// TIA Portal V17 export
// export: Created 2025-07-01T09:58:36.5371957Z, ExportSetting WithDefaults, DisplayName Totally Integrated Automation Portal, DisplayVersion V17 Update 8, DisplayName TIA Portal Openness, DisplayVersion V17 Update 8, DisplayName TIA Portal Version Control Interface, DisplayVersion V17, DisplayName SINAMICS Startdrive Advanced, DisplayVersion V17 SP2, DisplayName SINAMICS Startdrive G110M, G120, G120C, G120D, G120P, G115D, DisplayVersion V17 SP2, DisplayName SINAMICS Startdrive G130, G150, S120, S150, SINAMICS MV, S210, DisplayVersion V17 SP2, DisplayName STEP 7 Professional, DisplayVersion V17 Update 8, DisplayName SINUMERIK ONE STEP 7 Toolbox, DisplayVersion V17 Update 12, DisplayName SINUMERIK ONE PLC Basic Program Plus, DisplayVersion V17 Update 12, DisplayName SINUMERIK 840D sl STEP 7 Toolbox, DisplayVersion V17 Update 12, DisplayName STEP 7 Safety, DisplayVersion V17 Update 6, DisplayName WinCC Advanced, DisplayVersion V17 Update 8
FUNCTION "FC356_NCK_M_CH4_UNIT_2_STA_0" : Void   // FC356, LAD
TITLE = Channel 1 data
{ S7_Optimized_Access := 'FALSE' }
AUTHOR : ETXETAR
VERSION : 1.0
// stored: AutoNumber false, IsIECCheckEnabled false, SetENOAutomatically false, UDAEnableTagReadback false
   VAR_TEMP
      auxm3 : Bool;
      auxm5 : Bool;
   END_VAR
   VAR_TEMP   // added for the SCL form of the ladder/FBD networks
      _w1 : Bool;
      _w2 : Bool;
   END_VAR
BEGIN

REGION Network 1: CALL FB331 M CODE EXTENDED CH1 / M CODE EXTENDED CHANNEL 1
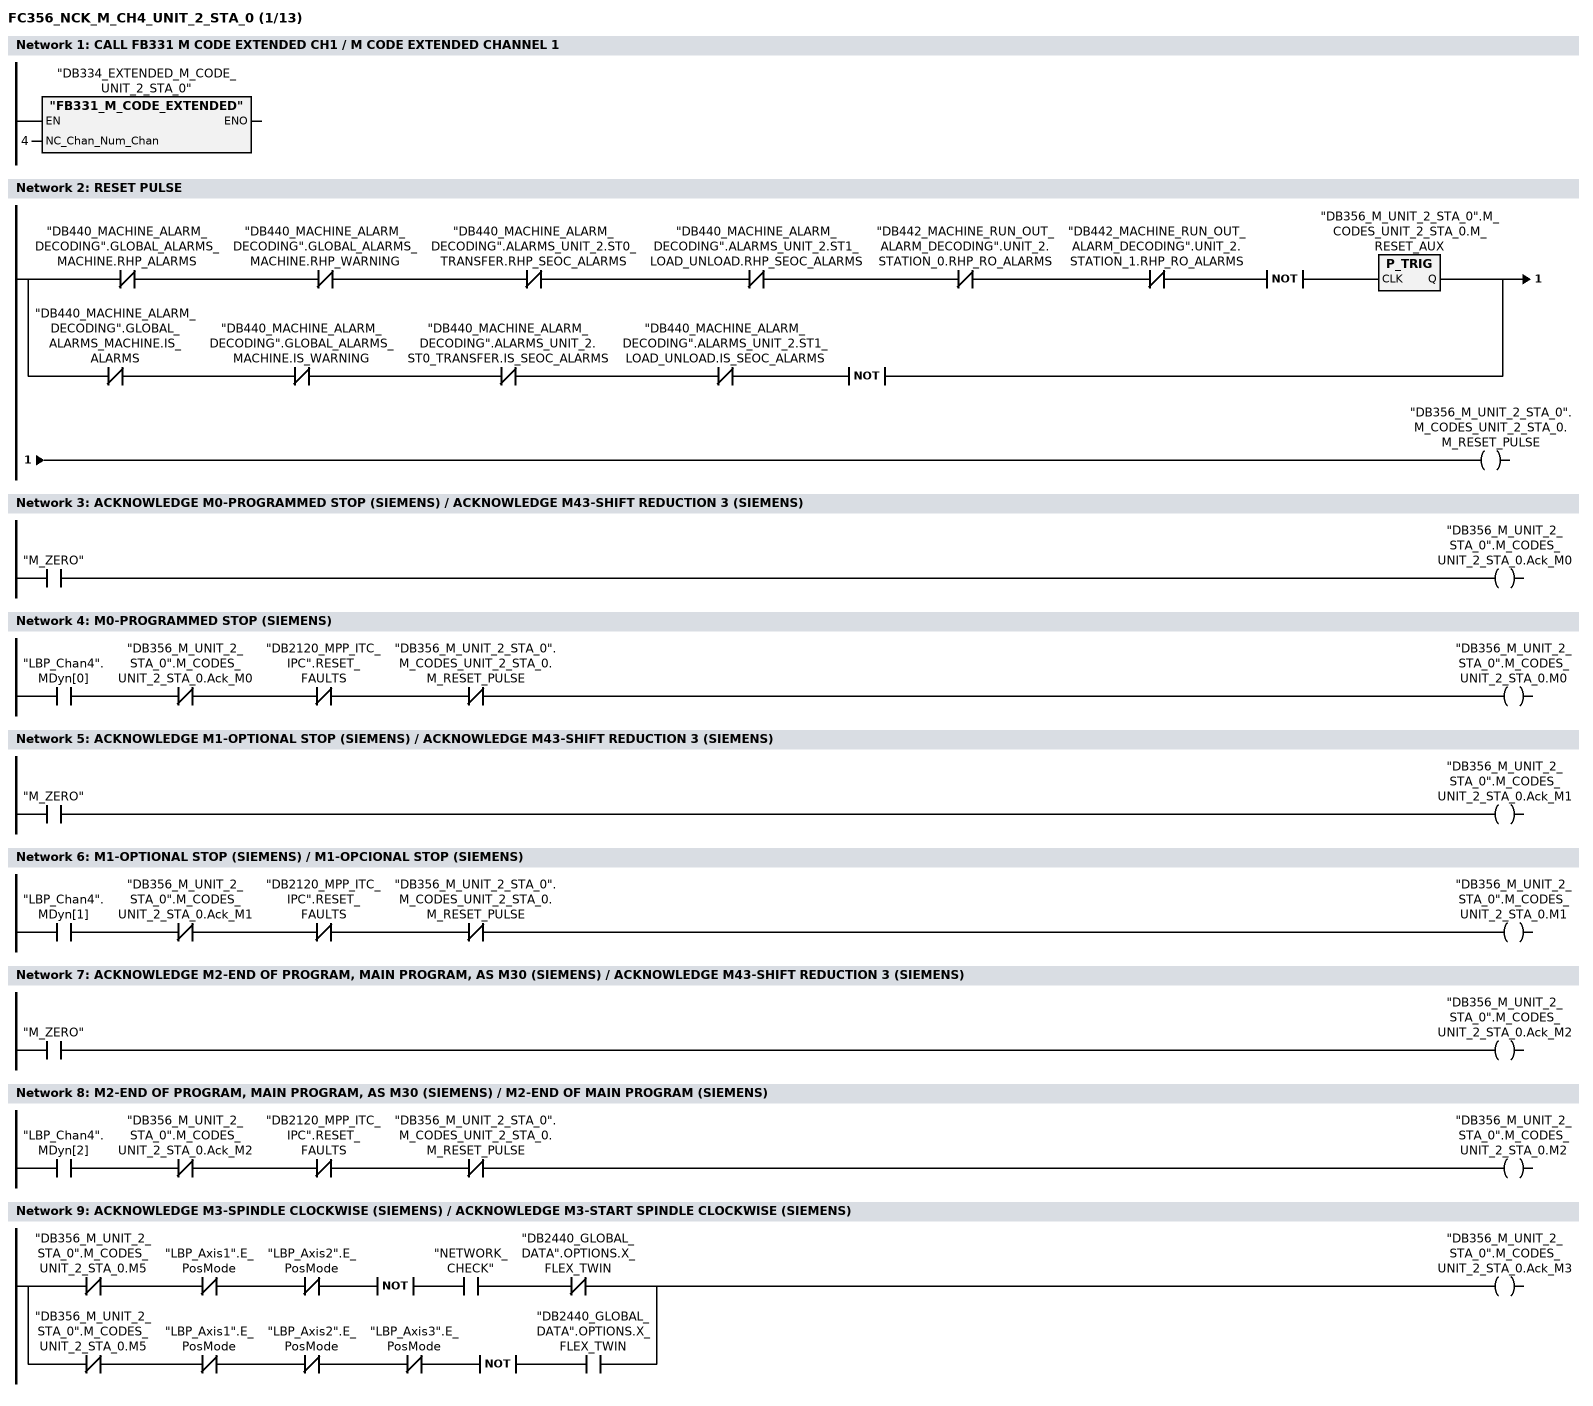
   RUNG wire#powerrail
      "DB334_EXTENDED_M_CODE_UNIT_2_STA_0"(NC_Chan_Num_Chan := 4)
   END_RUNG
   // the same network as SCL:
   "DB334_EXTENDED_M_CODE_UNIT_2_STA_0"(NC_Chan_Num_Chan := 4);   // "FB331_M_CODE_EXTENDED"
END_REGION

REGION Network 2: RESET PULSE
   RUNG wire#powerrail
      I_Contact( "DB440_MACHINE_ALARM_DECODING".GLOBAL_ALARMS_MACHINE.RHP_ALARMS )
      I_Contact( "DB440_MACHINE_ALARM_DECODING".GLOBAL_ALARMS_MACHINE.RHP_WARNING )
      I_Contact( "DB440_MACHINE_ALARM_DECODING".ALARMS_UNIT_2.ST0_TRANSFER.RHP_SEOC_ALARMS )
      I_Contact( "DB440_MACHINE_ALARM_DECODING".ALARMS_UNIT_2.ST1_LOAD_UNLOAD.RHP_SEOC_ALARMS )
      I_Contact( "DB442_MACHINE_RUN_OUT_ALARM_DECODING".UNIT_2.STATION_0.RHP_RO_ALARMS )
      I_Contact( "DB442_MACHINE_RUN_OUT_ALARM_DECODING".UNIT_2.STATION_1.RHP_RO_ALARMS )
      Not()
      P_Trig( "DB356_M_UNIT_2_STA_0".M_CODES_UNIT_2_STA_0.M_RESET_AUX )
      wire#w1
      Coil( "DB356_M_UNIT_2_STA_0".M_CODES_UNIT_2_STA_0.M_RESET_PULSE )
   END_RUNG
   RUNG wire#powerrail
      I_Contact( "DB440_MACHINE_ALARM_DECODING".GLOBAL_ALARMS_MACHINE.IS_ALARMS )
      I_Contact( "DB440_MACHINE_ALARM_DECODING".GLOBAL_ALARMS_MACHINE.IS_WARNING )
      I_Contact( "DB440_MACHINE_ALARM_DECODING".ALARMS_UNIT_2.ST0_TRANSFER.IS_SEOC_ALARMS )
      I_Contact( "DB440_MACHINE_ALARM_DECODING".ALARMS_UNIT_2.ST1_LOAD_UNLOAD.IS_SEOC_ALARMS )
      Not()
   END_RUNG wire#w1
   // the same network as SCL:
   #_w1 := NOT (NOT "DB440_MACHINE_ALARM_DECODING".GLOBAL_ALARMS_MACHINE.RHP_ALARMS AND NOT "DB440_MACHINE_ALARM_DECODING".GLOBAL_ALARMS_MACHINE.RHP_WARNING AND NOT "DB440_MACHINE_ALARM_DECODING".ALARMS_UNIT_2.ST0_TRANSFER.RHP_SEOC_ALARMS AND NOT "DB440_MACHINE_ALARM_DECODING".ALARMS_UNIT_2.ST1_LOAD_UNLOAD.RHP_SEOC_ALARMS AND NOT "DB442_MACHINE_RUN_OUT_ALARM_DECODING".UNIT_2.STATION_0.RHP_RO_ALARMS AND NOT "DB442_MACHINE_RUN_OUT_ALARM_DECODING".UNIT_2.STATION_1.RHP_RO_ALARMS);
   #_w2 := #_w1 AND NOT "DB356_M_UNIT_2_STA_0".M_CODES_UNIT_2_STA_0.M_RESET_AUX;   // rising edge
   "DB356_M_UNIT_2_STA_0".M_CODES_UNIT_2_STA_0.M_RESET_AUX := #_w1;
   "DB356_M_UNIT_2_STA_0".M_CODES_UNIT_2_STA_0.M_RESET_PULSE := #_w2 OR NOT (NOT "DB440_MACHINE_ALARM_DECODING".GLOBAL_ALARMS_MACHINE.IS_ALARMS AND NOT "DB440_MACHINE_ALARM_DECODING".GLOBAL_ALARMS_MACHINE.IS_WARNING AND NOT "DB440_MACHINE_ALARM_DECODING".ALARMS_UNIT_2.ST0_TRANSFER.IS_SEOC_ALARMS AND NOT "DB440_MACHINE_ALARM_DECODING".ALARMS_UNIT_2.ST1_LOAD_UNLOAD.IS_SEOC_ALARMS);
END_REGION

REGION Network 3: ACKNOWLEDGE M0-PROGRAMMED STOP (SIEMENS) / ACKNOWLEDGE M43-SHIFT REDUCTION 3 (SIEMENS)
   RUNG wire#powerrail
      Contact( "M_ZERO" )
      Coil( "DB356_M_UNIT_2_STA_0".M_CODES_UNIT_2_STA_0.Ack_M0 )
   END_RUNG
   // the same network as SCL:
   "DB356_M_UNIT_2_STA_0".M_CODES_UNIT_2_STA_0.Ack_M0 := "M_ZERO";
END_REGION

REGION Network 4: M0-PROGRAMMED STOP (SIEMENS)
   RUNG wire#powerrail
      Contact( "LBP_Chan4".MDyn[0] )
      I_Contact( "DB356_M_UNIT_2_STA_0".M_CODES_UNIT_2_STA_0.Ack_M0 )
      I_Contact( "DB2120_MPP_ITC_IPC".RESET_FAULTS )
      I_Contact( "DB356_M_UNIT_2_STA_0".M_CODES_UNIT_2_STA_0.M_RESET_PULSE )
      Coil( "DB356_M_UNIT_2_STA_0".M_CODES_UNIT_2_STA_0.M0 )
   END_RUNG
   // the same network as SCL:
   "DB356_M_UNIT_2_STA_0".M_CODES_UNIT_2_STA_0.M0 := "LBP_Chan4".MDyn[0] AND NOT "DB356_M_UNIT_2_STA_0".M_CODES_UNIT_2_STA_0.Ack_M0 AND NOT "DB2120_MPP_ITC_IPC".RESET_FAULTS AND NOT "DB356_M_UNIT_2_STA_0".M_CODES_UNIT_2_STA_0.M_RESET_PULSE;
END_REGION

REGION Network 5: ACKNOWLEDGE M1-OPTIONAL STOP (SIEMENS) / ACKNOWLEDGE M43-SHIFT REDUCTION 3 (SIEMENS)
   RUNG wire#powerrail
      Contact( "M_ZERO" )
      Coil( "DB356_M_UNIT_2_STA_0".M_CODES_UNIT_2_STA_0.Ack_M1 )
   END_RUNG
   // the same network as SCL:
   "DB356_M_UNIT_2_STA_0".M_CODES_UNIT_2_STA_0.Ack_M1 := "M_ZERO";
END_REGION

REGION Network 6: M1-OPTIONAL STOP (SIEMENS) / M1-OPCIONAL STOP (SIEMENS)
   RUNG wire#powerrail
      Contact( "LBP_Chan4".MDyn[1] )
      I_Contact( "DB356_M_UNIT_2_STA_0".M_CODES_UNIT_2_STA_0.Ack_M1 )
      I_Contact( "DB2120_MPP_ITC_IPC".RESET_FAULTS )
      I_Contact( "DB356_M_UNIT_2_STA_0".M_CODES_UNIT_2_STA_0.M_RESET_PULSE )
      Coil( "DB356_M_UNIT_2_STA_0".M_CODES_UNIT_2_STA_0.M1 )
   END_RUNG
   // the same network as SCL:
   "DB356_M_UNIT_2_STA_0".M_CODES_UNIT_2_STA_0.M1 := "LBP_Chan4".MDyn[1] AND NOT "DB356_M_UNIT_2_STA_0".M_CODES_UNIT_2_STA_0.Ack_M1 AND NOT "DB2120_MPP_ITC_IPC".RESET_FAULTS AND NOT "DB356_M_UNIT_2_STA_0".M_CODES_UNIT_2_STA_0.M_RESET_PULSE;
END_REGION

REGION Network 7: ACKNOWLEDGE M2-END OF PROGRAM, MAIN PROGRAM, AS M30 (SIEMENS) / ACKNOWLEDGE M43-SHIFT REDUCTION 3 (SIEMENS)
   RUNG wire#powerrail
      Contact( "M_ZERO" )
      Coil( "DB356_M_UNIT_2_STA_0".M_CODES_UNIT_2_STA_0.Ack_M2 )
   END_RUNG
   // the same network as SCL:
   "DB356_M_UNIT_2_STA_0".M_CODES_UNIT_2_STA_0.Ack_M2 := "M_ZERO";
END_REGION

REGION Network 8: M2-END OF PROGRAM, MAIN PROGRAM, AS M30 (SIEMENS) / M2-END OF MAIN PROGRAM (SIEMENS)
   RUNG wire#powerrail
      Contact( "LBP_Chan4".MDyn[2] )
      I_Contact( "DB356_M_UNIT_2_STA_0".M_CODES_UNIT_2_STA_0.Ack_M2 )
      I_Contact( "DB2120_MPP_ITC_IPC".RESET_FAULTS )
      I_Contact( "DB356_M_UNIT_2_STA_0".M_CODES_UNIT_2_STA_0.M_RESET_PULSE )
      Coil( "DB356_M_UNIT_2_STA_0".M_CODES_UNIT_2_STA_0.M2 )
   END_RUNG
   // the same network as SCL:
   "DB356_M_UNIT_2_STA_0".M_CODES_UNIT_2_STA_0.M2 := "LBP_Chan4".MDyn[2] AND NOT "DB356_M_UNIT_2_STA_0".M_CODES_UNIT_2_STA_0.Ack_M2 AND NOT "DB2120_MPP_ITC_IPC".RESET_FAULTS AND NOT "DB356_M_UNIT_2_STA_0".M_CODES_UNIT_2_STA_0.M_RESET_PULSE;
END_REGION

REGION Network 9: ACKNOWLEDGE M3-SPINDLE CLOCKWISE (SIEMENS) / ACKNOWLEDGE M3-START SPINDLE CLOCKWISE (SIEMENS)
   RUNG wire#powerrail
      I_Contact( "DB356_M_UNIT_2_STA_0".M_CODES_UNIT_2_STA_0.M5 )
      I_Contact( "LBP_Axis1".E_PosMode )
      I_Contact( "LBP_Axis2".E_PosMode )
      Not()
      Contact( "NETWORK_CHECK" )
      I_Contact( "DB2440_GLOBAL_DATA".OPTIONS.X_FLEX_TWIN )
      wire#w1
      Coil( "DB356_M_UNIT_2_STA_0".M_CODES_UNIT_2_STA_0.Ack_M3 )
   END_RUNG
   RUNG wire#powerrail
      I_Contact( "DB356_M_UNIT_2_STA_0".M_CODES_UNIT_2_STA_0.M5 )
      I_Contact( "LBP_Axis1".E_PosMode )
      I_Contact( "LBP_Axis2".E_PosMode )
      I_Contact( "LBP_Axis3".E_PosMode )
      Not()
      Contact( "DB2440_GLOBAL_DATA".OPTIONS.X_FLEX_TWIN )
   END_RUNG wire#w1
   // the same network as SCL:
   "DB356_M_UNIT_2_STA_0".M_CODES_UNIT_2_STA_0.Ack_M3 := (NOT (NOT "DB356_M_UNIT_2_STA_0".M_CODES_UNIT_2_STA_0.M5 AND NOT "LBP_Axis1".E_PosMode AND NOT "LBP_Axis2".E_PosMode) AND "NETWORK_CHECK" AND NOT "DB2440_GLOBAL_DATA".OPTIONS.X_FLEX_TWIN) OR (NOT (NOT "DB356_M_UNIT_2_STA_0".M_CODES_UNIT_2_STA_0.M5 AND NOT "LBP_Axis1".E_PosMode AND NOT "LBP_Axis2".E_PosMode AND NOT "LBP_Axis3".E_PosMode) AND "DB2440_GLOBAL_DATA".OPTIONS.X_FLEX_TWIN);
END_REGION

REGION Network 10: M3-SPINDLE CLOCKWISE AUXILIARY (SIEMENS) / Extended address M function 1 (16 bit INT)
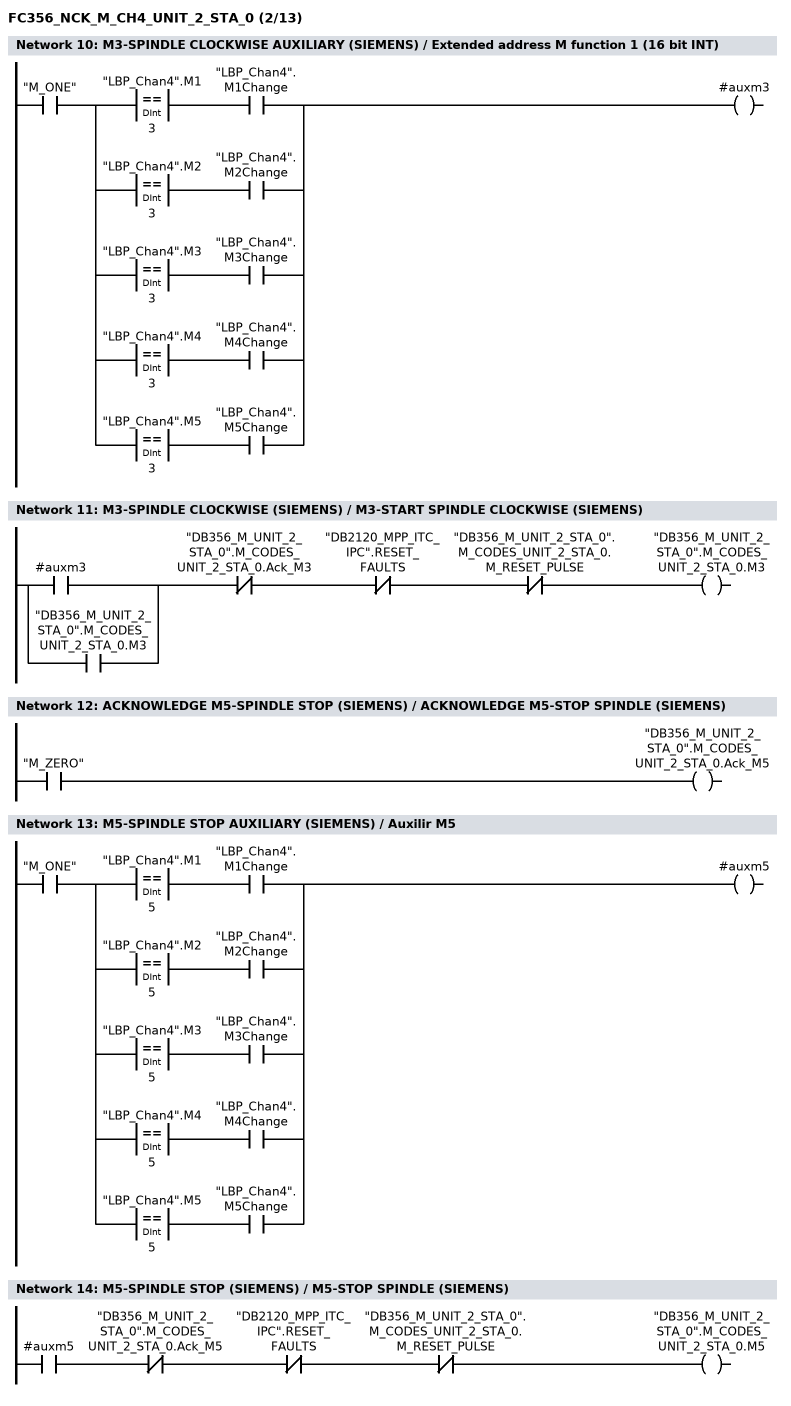
   RUNG wire#powerrail
      Contact( "M_ONE" )
      wire#w1
      { S7_Templates := "SrcType := DInt" } EQ_Contact(in1 := "LBP_Chan4".M1, in2 := 3)
      Contact( "LBP_Chan4".M1Change )
      wire#w2
      Coil( #auxm3 )
   END_RUNG
   RUNG wire#w1
      { S7_Templates := "SrcType := DInt" } EQ_Contact(in1 := "LBP_Chan4".M2, in2 := 3)
      Contact( "LBP_Chan4".M2Change )
   END_RUNG wire#w2
   RUNG wire#w1
      { S7_Templates := "SrcType := DInt" } EQ_Contact(in1 := "LBP_Chan4".M3, in2 := 3)
      Contact( "LBP_Chan4".M3Change )
   END_RUNG wire#w2
   RUNG wire#w1
      { S7_Templates := "SrcType := DInt" } EQ_Contact(in1 := "LBP_Chan4".M4, in2 := 3)
      Contact( "LBP_Chan4".M4Change )
   END_RUNG wire#w2
   RUNG wire#w1
      { S7_Templates := "SrcType := DInt" } EQ_Contact(in1 := "LBP_Chan4".M5, in2 := 3)
      Contact( "LBP_Chan4".M5Change )
   END_RUNG wire#w2
   // the same network as SCL:
   #auxm3 := "M_ONE" AND ((("LBP_Chan4".M1 = 3) AND "LBP_Chan4".M1Change) OR (("LBP_Chan4".M2 = 3) AND "LBP_Chan4".M2Change) OR (("LBP_Chan4".M3 = 3) AND "LBP_Chan4".M3Change) OR (("LBP_Chan4".M4 = 3) AND "LBP_Chan4".M4Change) OR (("LBP_Chan4".M5 = 3) AND "LBP_Chan4".M5Change));
END_REGION

REGION Network 11: M3-SPINDLE CLOCKWISE (SIEMENS) / M3-START SPINDLE CLOCKWISE (SIEMENS)
   RUNG wire#powerrail
      Contact( #auxm3 )
      wire#w1
      I_Contact( "DB356_M_UNIT_2_STA_0".M_CODES_UNIT_2_STA_0.Ack_M3 )
      I_Contact( "DB2120_MPP_ITC_IPC".RESET_FAULTS )
      I_Contact( "DB356_M_UNIT_2_STA_0".M_CODES_UNIT_2_STA_0.M_RESET_PULSE )
      Coil( "DB356_M_UNIT_2_STA_0".M_CODES_UNIT_2_STA_0.M3 )
   END_RUNG
   RUNG wire#powerrail
      Contact( "DB356_M_UNIT_2_STA_0".M_CODES_UNIT_2_STA_0.M3 )
   END_RUNG wire#w1
   // the same network as SCL:
   "DB356_M_UNIT_2_STA_0".M_CODES_UNIT_2_STA_0.M3 := (#auxm3 OR "DB356_M_UNIT_2_STA_0".M_CODES_UNIT_2_STA_0.M3) AND NOT "DB356_M_UNIT_2_STA_0".M_CODES_UNIT_2_STA_0.Ack_M3 AND NOT "DB2120_MPP_ITC_IPC".RESET_FAULTS AND NOT "DB356_M_UNIT_2_STA_0".M_CODES_UNIT_2_STA_0.M_RESET_PULSE;
END_REGION

REGION Network 12: ACKNOWLEDGE M5-SPINDLE STOP (SIEMENS) / ACKNOWLEDGE M5-STOP SPINDLE (SIEMENS)
   RUNG wire#powerrail
      Contact( "M_ZERO" )
      Coil( "DB356_M_UNIT_2_STA_0".M_CODES_UNIT_2_STA_0.Ack_M5 )
   END_RUNG
   // the same network as SCL:
   "DB356_M_UNIT_2_STA_0".M_CODES_UNIT_2_STA_0.Ack_M5 := "M_ZERO";
END_REGION

REGION Network 13: M5-SPINDLE STOP AUXILIARY (SIEMENS) / Auxilir M5
   RUNG wire#powerrail
      Contact( "M_ONE" )
      wire#w1
      { S7_Templates := "SrcType := DInt" } EQ_Contact(in1 := "LBP_Chan4".M1, in2 := 5)
      Contact( "LBP_Chan4".M1Change )
      wire#w2
      Coil( #auxm5 )
   END_RUNG
   RUNG wire#w1
      { S7_Templates := "SrcType := DInt" } EQ_Contact(in1 := "LBP_Chan4".M2, in2 := 5)
      Contact( "LBP_Chan4".M2Change )
   END_RUNG wire#w2
   RUNG wire#w1
      { S7_Templates := "SrcType := DInt" } EQ_Contact(in1 := "LBP_Chan4".M3, in2 := 5)
      Contact( "LBP_Chan4".M3Change )
   END_RUNG wire#w2
   RUNG wire#w1
      { S7_Templates := "SrcType := DInt" } EQ_Contact(in1 := "LBP_Chan4".M4, in2 := 5)
      Contact( "LBP_Chan4".M4Change )
   END_RUNG wire#w2
   RUNG wire#w1
      { S7_Templates := "SrcType := DInt" } EQ_Contact(in1 := "LBP_Chan4".M5, in2 := 5)
      Contact( "LBP_Chan4".M5Change )
   END_RUNG wire#w2
   // the same network as SCL:
   #auxm5 := "M_ONE" AND ((("LBP_Chan4".M1 = 5) AND "LBP_Chan4".M1Change) OR (("LBP_Chan4".M2 = 5) AND "LBP_Chan4".M2Change) OR (("LBP_Chan4".M3 = 5) AND "LBP_Chan4".M3Change) OR (("LBP_Chan4".M4 = 5) AND "LBP_Chan4".M4Change) OR (("LBP_Chan4".M5 = 5) AND "LBP_Chan4".M5Change));
END_REGION

REGION Network 14: M5-SPINDLE STOP (SIEMENS) / M5-STOP SPINDLE (SIEMENS)
   RUNG wire#powerrail
      Contact( #auxm5 )
      I_Contact( "DB356_M_UNIT_2_STA_0".M_CODES_UNIT_2_STA_0.Ack_M5 )
      I_Contact( "DB2120_MPP_ITC_IPC".RESET_FAULTS )
      I_Contact( "DB356_M_UNIT_2_STA_0".M_CODES_UNIT_2_STA_0.M_RESET_PULSE )
      Coil( "DB356_M_UNIT_2_STA_0".M_CODES_UNIT_2_STA_0.M5 )
   END_RUNG
   // the same network as SCL:
   "DB356_M_UNIT_2_STA_0".M_CODES_UNIT_2_STA_0.M5 := #auxm5 AND NOT "DB356_M_UNIT_2_STA_0".M_CODES_UNIT_2_STA_0.Ack_M5 AND NOT "DB2120_MPP_ITC_IPC".RESET_FAULTS AND NOT "DB356_M_UNIT_2_STA_0".M_CODES_UNIT_2_STA_0.M_RESET_PULSE;
END_REGION

REGION Network 15: M FUNCTIONS (DINT)
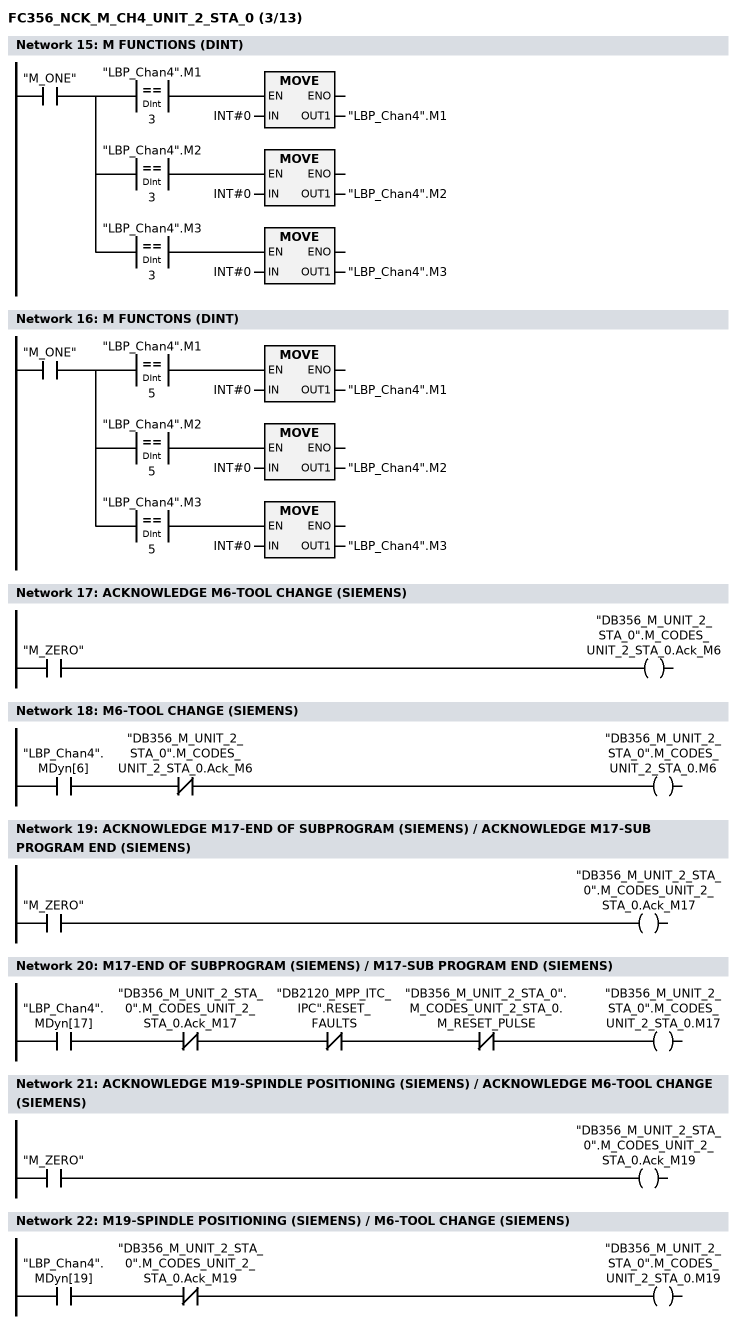
   RUNG wire#powerrail
      Contact( "M_ONE" )
      wire#w1
      { S7_Templates := "SrcType := DInt" } EQ_Contact(in1 := "LBP_Chan4".M1, in2 := 3)
      { S7_GenerateENO := "TRUE" } Move(in := INT#0, out1 => "LBP_Chan4".M1)
   END_RUNG
   RUNG wire#w1
      { S7_Templates := "SrcType := DInt" } EQ_Contact(in1 := "LBP_Chan4".M2, in2 := 3)
      { S7_GenerateENO := "TRUE" } Move(in := INT#0, out1 => "LBP_Chan4".M2)
   END_RUNG
   RUNG wire#w1
      { S7_Templates := "SrcType := DInt" } EQ_Contact(in1 := "LBP_Chan4".M3, in2 := 3)
      { S7_GenerateENO := "TRUE" } Move(in := INT#0, out1 => "LBP_Chan4".M3)
   END_RUNG
   // the same network as SCL:
   IF "M_ONE" AND ("LBP_Chan4".M1 = 3) THEN "LBP_Chan4".M1 := INT#0; END_IF;
   IF "M_ONE" AND ("LBP_Chan4".M2 = 3) THEN "LBP_Chan4".M2 := INT#0; END_IF;
   IF "M_ONE" AND ("LBP_Chan4".M3 = 3) THEN "LBP_Chan4".M3 := INT#0; END_IF;
END_REGION

REGION Network 16: M FUNCTONS (DINT)
   RUNG wire#powerrail
      Contact( "M_ONE" )
      wire#w1
      { S7_Templates := "SrcType := DInt" } EQ_Contact(in1 := "LBP_Chan4".M1, in2 := 5)
      { S7_GenerateENO := "TRUE" } Move(in := INT#0, out1 => "LBP_Chan4".M1)
   END_RUNG
   RUNG wire#w1
      { S7_Templates := "SrcType := DInt" } EQ_Contact(in1 := "LBP_Chan4".M2, in2 := 5)
      { S7_GenerateENO := "TRUE" } Move(in := INT#0, out1 => "LBP_Chan4".M2)
   END_RUNG
   RUNG wire#w1
      { S7_Templates := "SrcType := DInt" } EQ_Contact(in1 := "LBP_Chan4".M3, in2 := 5)
      { S7_GenerateENO := "TRUE" } Move(in := INT#0, out1 => "LBP_Chan4".M3)
   END_RUNG
   // the same network as SCL:
   IF "M_ONE" AND ("LBP_Chan4".M1 = 5) THEN "LBP_Chan4".M1 := INT#0; END_IF;
   IF "M_ONE" AND ("LBP_Chan4".M2 = 5) THEN "LBP_Chan4".M2 := INT#0; END_IF;
   IF "M_ONE" AND ("LBP_Chan4".M3 = 5) THEN "LBP_Chan4".M3 := INT#0; END_IF;
END_REGION

REGION Network 17: ACKNOWLEDGE M6-TOOL CHANGE (SIEMENS)
   RUNG wire#powerrail
      Contact( "M_ZERO" )
      Coil( "DB356_M_UNIT_2_STA_0".M_CODES_UNIT_2_STA_0.Ack_M6 )
   END_RUNG
   // the same network as SCL:
   "DB356_M_UNIT_2_STA_0".M_CODES_UNIT_2_STA_0.Ack_M6 := "M_ZERO";
END_REGION

REGION Network 18: M6-TOOL CHANGE (SIEMENS)
   RUNG wire#powerrail
      Contact( "LBP_Chan4".MDyn[6] )
      I_Contact( "DB356_M_UNIT_2_STA_0".M_CODES_UNIT_2_STA_0.Ack_M6 )
      Coil( "DB356_M_UNIT_2_STA_0".M_CODES_UNIT_2_STA_0.M6 )
   END_RUNG
   // the same network as SCL:
   "DB356_M_UNIT_2_STA_0".M_CODES_UNIT_2_STA_0.M6 := "LBP_Chan4".MDyn[6] AND NOT "DB356_M_UNIT_2_STA_0".M_CODES_UNIT_2_STA_0.Ack_M6;
END_REGION

REGION Network 19: ACKNOWLEDGE M17-END OF SUBPROGRAM (SIEMENS) / ACKNOWLEDGE M17-SUB PROGRAM END (SIEMENS)
   RUNG wire#powerrail
      Contact( "M_ZERO" )
      Coil( "DB356_M_UNIT_2_STA_0".M_CODES_UNIT_2_STA_0.Ack_M17 )
   END_RUNG
   // the same network as SCL:
   "DB356_M_UNIT_2_STA_0".M_CODES_UNIT_2_STA_0.Ack_M17 := "M_ZERO";
END_REGION

REGION Network 20: M17-END OF SUBPROGRAM (SIEMENS) / M17-SUB PROGRAM END (SIEMENS)
   RUNG wire#powerrail
      Contact( "LBP_Chan4".MDyn[17] )
      I_Contact( "DB356_M_UNIT_2_STA_0".M_CODES_UNIT_2_STA_0.Ack_M17 )
      I_Contact( "DB2120_MPP_ITC_IPC".RESET_FAULTS )
      I_Contact( "DB356_M_UNIT_2_STA_0".M_CODES_UNIT_2_STA_0.M_RESET_PULSE )
      Coil( "DB356_M_UNIT_2_STA_0".M_CODES_UNIT_2_STA_0.M17 )
   END_RUNG
   // the same network as SCL:
   "DB356_M_UNIT_2_STA_0".M_CODES_UNIT_2_STA_0.M17 := "LBP_Chan4".MDyn[17] AND NOT "DB356_M_UNIT_2_STA_0".M_CODES_UNIT_2_STA_0.Ack_M17 AND NOT "DB2120_MPP_ITC_IPC".RESET_FAULTS AND NOT "DB356_M_UNIT_2_STA_0".M_CODES_UNIT_2_STA_0.M_RESET_PULSE;
END_REGION

REGION Network 21: ACKNOWLEDGE M19-SPINDLE POSITIONING (SIEMENS) / ACKNOWLEDGE M6-TOOL CHANGE (SIEMENS)
   RUNG wire#powerrail
      Contact( "M_ZERO" )
      Coil( "DB356_M_UNIT_2_STA_0".M_CODES_UNIT_2_STA_0.Ack_M19 )
   END_RUNG
   // the same network as SCL:
   "DB356_M_UNIT_2_STA_0".M_CODES_UNIT_2_STA_0.Ack_M19 := "M_ZERO";
END_REGION

REGION Network 22: M19-SPINDLE POSITIONING (SIEMENS) / M6-TOOL CHANGE (SIEMENS)
   RUNG wire#powerrail
      Contact( "LBP_Chan4".MDyn[19] )
      I_Contact( "DB356_M_UNIT_2_STA_0".M_CODES_UNIT_2_STA_0.Ack_M19 )
      Coil( "DB356_M_UNIT_2_STA_0".M_CODES_UNIT_2_STA_0.M19 )
   END_RUNG
   // the same network as SCL:
   "DB356_M_UNIT_2_STA_0".M_CODES_UNIT_2_STA_0.M19 := "LBP_Chan4".MDyn[19] AND NOT "DB356_M_UNIT_2_STA_0".M_CODES_UNIT_2_STA_0.Ack_M19;
END_REGION

REGION Network 23: ACKNOWLEDGE M20-FIXTURE 1 TOTAL FULL DEPTH / ACKNOWLEDGE M90-TOTAL FULL DEPTH
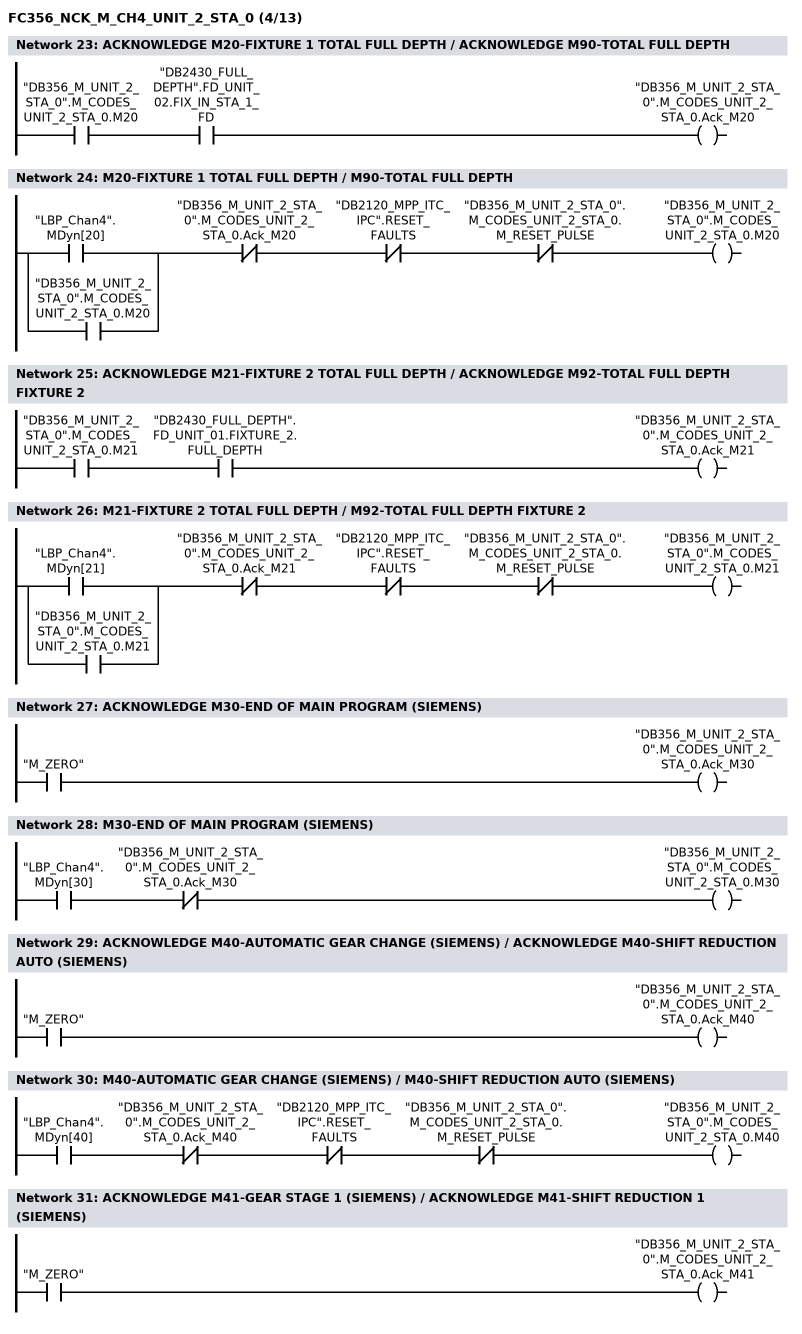
   RUNG wire#powerrail
      Contact( "DB356_M_UNIT_2_STA_0".M_CODES_UNIT_2_STA_0.M20 )
      Contact( "DB2430_FULL_DEPTH".FD_UNIT_02.FIX_IN_STA_1_FD )
      Coil( "DB356_M_UNIT_2_STA_0".M_CODES_UNIT_2_STA_0.Ack_M20 )
   END_RUNG
   // the same network as SCL:
   "DB356_M_UNIT_2_STA_0".M_CODES_UNIT_2_STA_0.Ack_M20 := "DB356_M_UNIT_2_STA_0".M_CODES_UNIT_2_STA_0.M20 AND "DB2430_FULL_DEPTH".FD_UNIT_02.FIX_IN_STA_1_FD;
END_REGION

REGION Network 24: M20-FIXTURE 1 TOTAL FULL DEPTH / M90-TOTAL FULL DEPTH
   RUNG wire#powerrail
      Contact( "LBP_Chan4".MDyn[20] )
      wire#w1
      I_Contact( "DB356_M_UNIT_2_STA_0".M_CODES_UNIT_2_STA_0.Ack_M20 )
      I_Contact( "DB2120_MPP_ITC_IPC".RESET_FAULTS )
      I_Contact( "DB356_M_UNIT_2_STA_0".M_CODES_UNIT_2_STA_0.M_RESET_PULSE )
      Coil( "DB356_M_UNIT_2_STA_0".M_CODES_UNIT_2_STA_0.M20 )
   END_RUNG
   RUNG wire#powerrail
      Contact( "DB356_M_UNIT_2_STA_0".M_CODES_UNIT_2_STA_0.M20 )
   END_RUNG wire#w1
   // the same network as SCL:
   "DB356_M_UNIT_2_STA_0".M_CODES_UNIT_2_STA_0.M20 := ("LBP_Chan4".MDyn[20] OR "DB356_M_UNIT_2_STA_0".M_CODES_UNIT_2_STA_0.M20) AND NOT "DB356_M_UNIT_2_STA_0".M_CODES_UNIT_2_STA_0.Ack_M20 AND NOT "DB2120_MPP_ITC_IPC".RESET_FAULTS AND NOT "DB356_M_UNIT_2_STA_0".M_CODES_UNIT_2_STA_0.M_RESET_PULSE;
END_REGION

REGION Network 25: ACKNOWLEDGE M21-FIXTURE 2 TOTAL FULL DEPTH / ACKNOWLEDGE M92-TOTAL FULL DEPTH FIXTURE 2
   RUNG wire#powerrail
      Contact( "DB356_M_UNIT_2_STA_0".M_CODES_UNIT_2_STA_0.M21 )
      Contact( "DB2430_FULL_DEPTH".FD_UNIT_01.FIXTURE_2.FULL_DEPTH )
      Coil( "DB356_M_UNIT_2_STA_0".M_CODES_UNIT_2_STA_0.Ack_M21 )
   END_RUNG
   // the same network as SCL:
   "DB356_M_UNIT_2_STA_0".M_CODES_UNIT_2_STA_0.Ack_M21 := "DB356_M_UNIT_2_STA_0".M_CODES_UNIT_2_STA_0.M21 AND "DB2430_FULL_DEPTH".FD_UNIT_01.FIXTURE_2.FULL_DEPTH;
END_REGION

REGION Network 26: M21-FIXTURE 2 TOTAL FULL DEPTH / M92-TOTAL FULL DEPTH FIXTURE 2
   RUNG wire#powerrail
      Contact( "LBP_Chan4".MDyn[21] )
      wire#w1
      I_Contact( "DB356_M_UNIT_2_STA_0".M_CODES_UNIT_2_STA_0.Ack_M21 )
      I_Contact( "DB2120_MPP_ITC_IPC".RESET_FAULTS )
      I_Contact( "DB356_M_UNIT_2_STA_0".M_CODES_UNIT_2_STA_0.M_RESET_PULSE )
      Coil( "DB356_M_UNIT_2_STA_0".M_CODES_UNIT_2_STA_0.M21 )
   END_RUNG
   RUNG wire#powerrail
      Contact( "DB356_M_UNIT_2_STA_0".M_CODES_UNIT_2_STA_0.M21 )
   END_RUNG wire#w1
   // the same network as SCL:
   "DB356_M_UNIT_2_STA_0".M_CODES_UNIT_2_STA_0.M21 := ("LBP_Chan4".MDyn[21] OR "DB356_M_UNIT_2_STA_0".M_CODES_UNIT_2_STA_0.M21) AND NOT "DB356_M_UNIT_2_STA_0".M_CODES_UNIT_2_STA_0.Ack_M21 AND NOT "DB2120_MPP_ITC_IPC".RESET_FAULTS AND NOT "DB356_M_UNIT_2_STA_0".M_CODES_UNIT_2_STA_0.M_RESET_PULSE;
END_REGION

REGION Network 27: ACKNOWLEDGE M30-END OF MAIN PROGRAM (SIEMENS)
   RUNG wire#powerrail
      Contact( "M_ZERO" )
      Coil( "DB356_M_UNIT_2_STA_0".M_CODES_UNIT_2_STA_0.Ack_M30 )
   END_RUNG
   // the same network as SCL:
   "DB356_M_UNIT_2_STA_0".M_CODES_UNIT_2_STA_0.Ack_M30 := "M_ZERO";
END_REGION

REGION Network 28: M30-END OF MAIN PROGRAM (SIEMENS)
   RUNG wire#powerrail
      Contact( "LBP_Chan4".MDyn[30] )
      I_Contact( "DB356_M_UNIT_2_STA_0".M_CODES_UNIT_2_STA_0.Ack_M30 )
      Coil( "DB356_M_UNIT_2_STA_0".M_CODES_UNIT_2_STA_0.M30 )
   END_RUNG
   // the same network as SCL:
   "DB356_M_UNIT_2_STA_0".M_CODES_UNIT_2_STA_0.M30 := "LBP_Chan4".MDyn[30] AND NOT "DB356_M_UNIT_2_STA_0".M_CODES_UNIT_2_STA_0.Ack_M30;
END_REGION

REGION Network 29: ACKNOWLEDGE M40-AUTOMATIC GEAR CHANGE (SIEMENS) / ACKNOWLEDGE M40-SHIFT REDUCTION AUTO (SIEMENS)
   RUNG wire#powerrail
      Contact( "M_ZERO" )
      Coil( "DB356_M_UNIT_2_STA_0".M_CODES_UNIT_2_STA_0.Ack_M40 )
   END_RUNG
   // the same network as SCL:
   "DB356_M_UNIT_2_STA_0".M_CODES_UNIT_2_STA_0.Ack_M40 := "M_ZERO";
END_REGION

REGION Network 30: M40-AUTOMATIC GEAR CHANGE (SIEMENS) / M40-SHIFT REDUCTION AUTO (SIEMENS)
   RUNG wire#powerrail
      Contact( "LBP_Chan4".MDyn[40] )
      I_Contact( "DB356_M_UNIT_2_STA_0".M_CODES_UNIT_2_STA_0.Ack_M40 )
      I_Contact( "DB2120_MPP_ITC_IPC".RESET_FAULTS )
      I_Contact( "DB356_M_UNIT_2_STA_0".M_CODES_UNIT_2_STA_0.M_RESET_PULSE )
      Coil( "DB356_M_UNIT_2_STA_0".M_CODES_UNIT_2_STA_0.M40 )
   END_RUNG
   // the same network as SCL:
   "DB356_M_UNIT_2_STA_0".M_CODES_UNIT_2_STA_0.M40 := "LBP_Chan4".MDyn[40] AND NOT "DB356_M_UNIT_2_STA_0".M_CODES_UNIT_2_STA_0.Ack_M40 AND NOT "DB2120_MPP_ITC_IPC".RESET_FAULTS AND NOT "DB356_M_UNIT_2_STA_0".M_CODES_UNIT_2_STA_0.M_RESET_PULSE;
END_REGION

REGION Network 31: ACKNOWLEDGE M41-GEAR STAGE 1 (SIEMENS) / ACKNOWLEDGE M41-SHIFT REDUCTION 1 (SIEMENS)
   RUNG wire#powerrail
      Contact( "M_ZERO" )
      Coil( "DB356_M_UNIT_2_STA_0".M_CODES_UNIT_2_STA_0.Ack_M41 )
   END_RUNG
   // the same network as SCL:
   "DB356_M_UNIT_2_STA_0".M_CODES_UNIT_2_STA_0.Ack_M41 := "M_ZERO";
END_REGION

REGION Network 32: M41-GEAR STAGE 1 (SIEMENS) / M41-SHIFT REDUCTION 1 (SIEMENS)
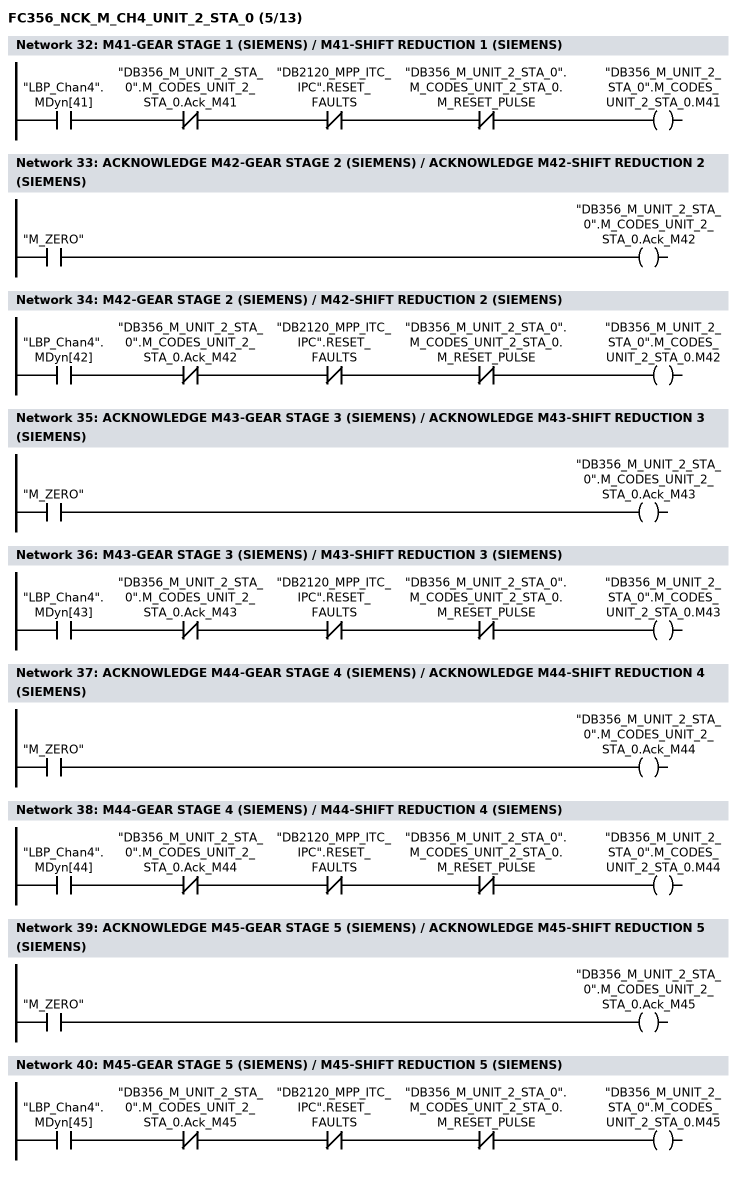
   RUNG wire#powerrail
      Contact( "LBP_Chan4".MDyn[41] )
      I_Contact( "DB356_M_UNIT_2_STA_0".M_CODES_UNIT_2_STA_0.Ack_M41 )
      I_Contact( "DB2120_MPP_ITC_IPC".RESET_FAULTS )
      I_Contact( "DB356_M_UNIT_2_STA_0".M_CODES_UNIT_2_STA_0.M_RESET_PULSE )
      Coil( "DB356_M_UNIT_2_STA_0".M_CODES_UNIT_2_STA_0.M41 )
   END_RUNG
   // the same network as SCL:
   "DB356_M_UNIT_2_STA_0".M_CODES_UNIT_2_STA_0.M41 := "LBP_Chan4".MDyn[41] AND NOT "DB356_M_UNIT_2_STA_0".M_CODES_UNIT_2_STA_0.Ack_M41 AND NOT "DB2120_MPP_ITC_IPC".RESET_FAULTS AND NOT "DB356_M_UNIT_2_STA_0".M_CODES_UNIT_2_STA_0.M_RESET_PULSE;
END_REGION

REGION Network 33: ACKNOWLEDGE M42-GEAR STAGE 2 (SIEMENS) / ACKNOWLEDGE M42-SHIFT REDUCTION 2 (SIEMENS)
   RUNG wire#powerrail
      Contact( "M_ZERO" )
      Coil( "DB356_M_UNIT_2_STA_0".M_CODES_UNIT_2_STA_0.Ack_M42 )
   END_RUNG
   // the same network as SCL:
   "DB356_M_UNIT_2_STA_0".M_CODES_UNIT_2_STA_0.Ack_M42 := "M_ZERO";
END_REGION

REGION Network 34: M42-GEAR STAGE 2 (SIEMENS) / M42-SHIFT REDUCTION 2 (SIEMENS)
   RUNG wire#powerrail
      Contact( "LBP_Chan4".MDyn[42] )
      I_Contact( "DB356_M_UNIT_2_STA_0".M_CODES_UNIT_2_STA_0.Ack_M42 )
      I_Contact( "DB2120_MPP_ITC_IPC".RESET_FAULTS )
      I_Contact( "DB356_M_UNIT_2_STA_0".M_CODES_UNIT_2_STA_0.M_RESET_PULSE )
      Coil( "DB356_M_UNIT_2_STA_0".M_CODES_UNIT_2_STA_0.M42 )
   END_RUNG
   // the same network as SCL:
   "DB356_M_UNIT_2_STA_0".M_CODES_UNIT_2_STA_0.M42 := "LBP_Chan4".MDyn[42] AND NOT "DB356_M_UNIT_2_STA_0".M_CODES_UNIT_2_STA_0.Ack_M42 AND NOT "DB2120_MPP_ITC_IPC".RESET_FAULTS AND NOT "DB356_M_UNIT_2_STA_0".M_CODES_UNIT_2_STA_0.M_RESET_PULSE;
END_REGION

REGION Network 35: ACKNOWLEDGE M43-GEAR STAGE 3 (SIEMENS) / ACKNOWLEDGE M43-SHIFT REDUCTION 3 (SIEMENS)
   RUNG wire#powerrail
      Contact( "M_ZERO" )
      Coil( "DB356_M_UNIT_2_STA_0".M_CODES_UNIT_2_STA_0.Ack_M43 )
   END_RUNG
   // the same network as SCL:
   "DB356_M_UNIT_2_STA_0".M_CODES_UNIT_2_STA_0.Ack_M43 := "M_ZERO";
END_REGION

REGION Network 36: M43-GEAR STAGE 3 (SIEMENS) / M43-SHIFT REDUCTION 3 (SIEMENS)
   RUNG wire#powerrail
      Contact( "LBP_Chan4".MDyn[43] )
      I_Contact( "DB356_M_UNIT_2_STA_0".M_CODES_UNIT_2_STA_0.Ack_M43 )
      I_Contact( "DB2120_MPP_ITC_IPC".RESET_FAULTS )
      I_Contact( "DB356_M_UNIT_2_STA_0".M_CODES_UNIT_2_STA_0.M_RESET_PULSE )
      Coil( "DB356_M_UNIT_2_STA_0".M_CODES_UNIT_2_STA_0.M43 )
   END_RUNG
   // the same network as SCL:
   "DB356_M_UNIT_2_STA_0".M_CODES_UNIT_2_STA_0.M43 := "LBP_Chan4".MDyn[43] AND NOT "DB356_M_UNIT_2_STA_0".M_CODES_UNIT_2_STA_0.Ack_M43 AND NOT "DB2120_MPP_ITC_IPC".RESET_FAULTS AND NOT "DB356_M_UNIT_2_STA_0".M_CODES_UNIT_2_STA_0.M_RESET_PULSE;
END_REGION

REGION Network 37: ACKNOWLEDGE M44-GEAR STAGE 4 (SIEMENS) / ACKNOWLEDGE M44-SHIFT REDUCTION 4 (SIEMENS)
   RUNG wire#powerrail
      Contact( "M_ZERO" )
      Coil( "DB356_M_UNIT_2_STA_0".M_CODES_UNIT_2_STA_0.Ack_M44 )
   END_RUNG
   // the same network as SCL:
   "DB356_M_UNIT_2_STA_0".M_CODES_UNIT_2_STA_0.Ack_M44 := "M_ZERO";
END_REGION

REGION Network 38: M44-GEAR STAGE 4 (SIEMENS) / M44-SHIFT REDUCTION 4 (SIEMENS)
   RUNG wire#powerrail
      Contact( "LBP_Chan4".MDyn[44] )
      I_Contact( "DB356_M_UNIT_2_STA_0".M_CODES_UNIT_2_STA_0.Ack_M44 )
      I_Contact( "DB2120_MPP_ITC_IPC".RESET_FAULTS )
      I_Contact( "DB356_M_UNIT_2_STA_0".M_CODES_UNIT_2_STA_0.M_RESET_PULSE )
      Coil( "DB356_M_UNIT_2_STA_0".M_CODES_UNIT_2_STA_0.M44 )
   END_RUNG
   // the same network as SCL:
   "DB356_M_UNIT_2_STA_0".M_CODES_UNIT_2_STA_0.M44 := "LBP_Chan4".MDyn[44] AND NOT "DB356_M_UNIT_2_STA_0".M_CODES_UNIT_2_STA_0.Ack_M44 AND NOT "DB2120_MPP_ITC_IPC".RESET_FAULTS AND NOT "DB356_M_UNIT_2_STA_0".M_CODES_UNIT_2_STA_0.M_RESET_PULSE;
END_REGION

REGION Network 39: ACKNOWLEDGE M45-GEAR STAGE 5 (SIEMENS) / ACKNOWLEDGE M45-SHIFT REDUCTION 5 (SIEMENS)
   RUNG wire#powerrail
      Contact( "M_ZERO" )
      Coil( "DB356_M_UNIT_2_STA_0".M_CODES_UNIT_2_STA_0.Ack_M45 )
   END_RUNG
   // the same network as SCL:
   "DB356_M_UNIT_2_STA_0".M_CODES_UNIT_2_STA_0.Ack_M45 := "M_ZERO";
END_REGION

REGION Network 40: M45-GEAR STAGE 5 (SIEMENS) / M45-SHIFT REDUCTION 5 (SIEMENS)
   RUNG wire#powerrail
      Contact( "LBP_Chan4".MDyn[45] )
      I_Contact( "DB356_M_UNIT_2_STA_0".M_CODES_UNIT_2_STA_0.Ack_M45 )
      I_Contact( "DB2120_MPP_ITC_IPC".RESET_FAULTS )
      I_Contact( "DB356_M_UNIT_2_STA_0".M_CODES_UNIT_2_STA_0.M_RESET_PULSE )
      Coil( "DB356_M_UNIT_2_STA_0".M_CODES_UNIT_2_STA_0.M45 )
   END_RUNG
   // the same network as SCL:
   "DB356_M_UNIT_2_STA_0".M_CODES_UNIT_2_STA_0.M45 := "LBP_Chan4".MDyn[45] AND NOT "DB356_M_UNIT_2_STA_0".M_CODES_UNIT_2_STA_0.Ack_M45 AND NOT "DB2120_MPP_ITC_IPC".RESET_FAULTS AND NOT "DB356_M_UNIT_2_STA_0".M_CODES_UNIT_2_STA_0.M_RESET_PULSE;
END_REGION

REGION Network 41: ACKNOWLEDGE M50-LOAD PART FROM ROBOT (READ IN DISABLE)
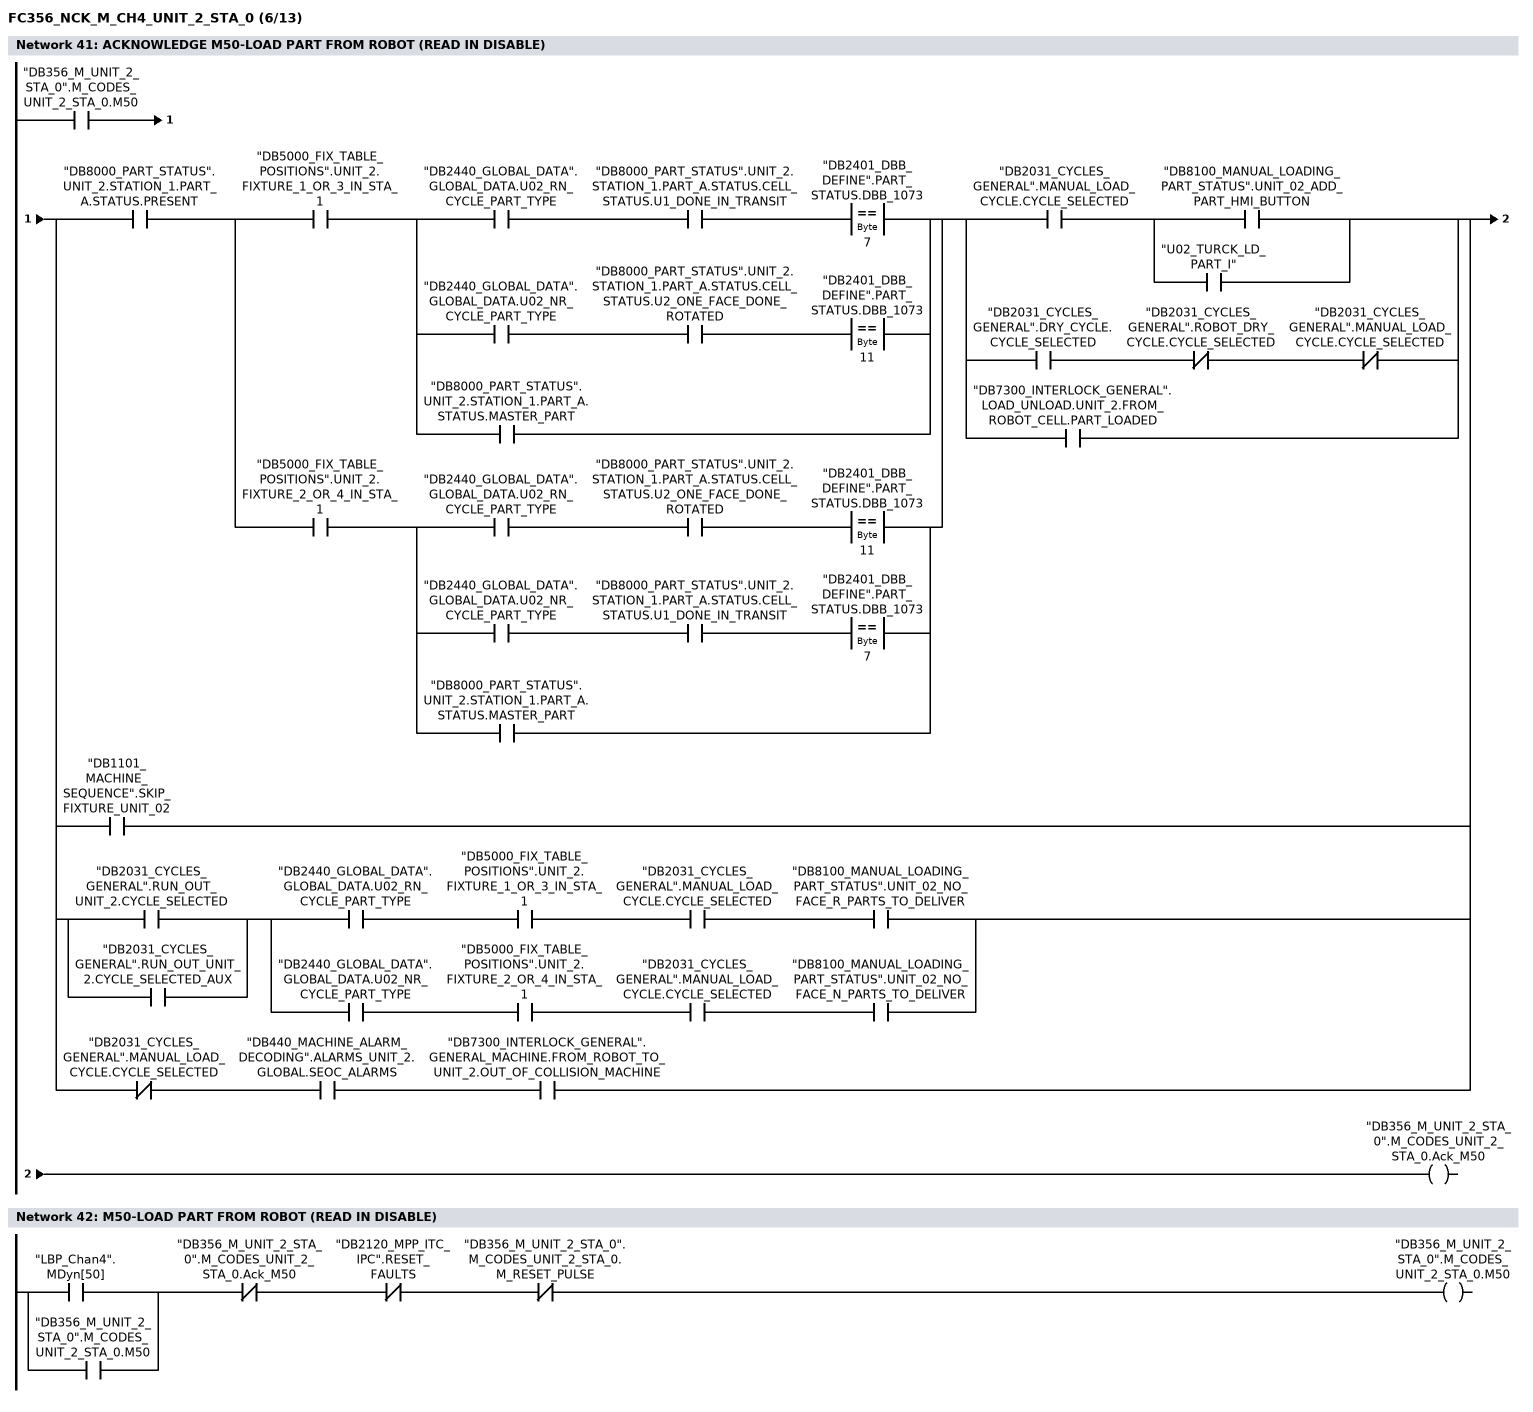
   RUNG wire#powerrail
      Contact( "DB356_M_UNIT_2_STA_0".M_CODES_UNIT_2_STA_0.M50 )
      wire#w1
      Contact( "DB8000_PART_STATUS".UNIT_2.STATION_1.PART_A.STATUS.PRESENT )
      wire#w2
      Contact( "DB5000_FIX_TABLE_POSITIONS".UNIT_2.FIXTURE_1_OR_3_IN_STA_1 )
      wire#w3
      Contact( "DB2440_GLOBAL_DATA".GLOBAL_DATA.U02_RN_CYCLE_PART_TYPE )
      Contact( "DB8000_PART_STATUS".UNIT_2.STATION_1.PART_A.STATUS.CELL_STATUS.U1_DONE_IN_TRANSIT )
      { S7_Templates := "SrcType := Byte" } EQ_Contact(in1 := "DB2401_DBB_DEFINE".PART_STATUS.DBB_1073, in2 := 7)
      wire#w4
      Contact( "DB2031_CYCLES_GENERAL".MANUAL_LOAD_CYCLE.CYCLE_SELECTED )
      wire#w6
      Contact( "DB8100_MANUAL_LOADING_PART_STATUS".UNIT_02_ADD_PART_HMI_BUTTON )
      wire#w7
      Coil( "DB356_M_UNIT_2_STA_0".M_CODES_UNIT_2_STA_0.Ack_M50 )
   END_RUNG
   RUNG wire#w3
      Contact( "DB2440_GLOBAL_DATA".GLOBAL_DATA.U02_NR_CYCLE_PART_TYPE )
      Contact( "DB8000_PART_STATUS".UNIT_2.STATION_1.PART_A.STATUS.CELL_STATUS.U2_ONE_FACE_DONE_ROTATED )
      { S7_Templates := "SrcType := Byte" } EQ_Contact(in1 := "DB2401_DBB_DEFINE".PART_STATUS.DBB_1073, in2 := 11)
   END_RUNG wire#w4
   RUNG wire#w3
      Contact( "DB8000_PART_STATUS".UNIT_2.STATION_1.PART_A.STATUS.MASTER_PART )
   END_RUNG wire#w4
   RUNG wire#w2
      Contact( "DB5000_FIX_TABLE_POSITIONS".UNIT_2.FIXTURE_2_OR_4_IN_STA_1 )
      wire#w5
      Contact( "DB2440_GLOBAL_DATA".GLOBAL_DATA.U02_RN_CYCLE_PART_TYPE )
      Contact( "DB8000_PART_STATUS".UNIT_2.STATION_1.PART_A.STATUS.CELL_STATUS.U2_ONE_FACE_DONE_ROTATED )
      { S7_Templates := "SrcType := Byte" } EQ_Contact(in1 := "DB2401_DBB_DEFINE".PART_STATUS.DBB_1073, in2 := 11)
   END_RUNG wire#w4
   RUNG wire#w5
      Contact( "DB2440_GLOBAL_DATA".GLOBAL_DATA.U02_NR_CYCLE_PART_TYPE )
      Contact( "DB8000_PART_STATUS".UNIT_2.STATION_1.PART_A.STATUS.CELL_STATUS.U1_DONE_IN_TRANSIT )
      { S7_Templates := "SrcType := Byte" } EQ_Contact(in1 := "DB2401_DBB_DEFINE".PART_STATUS.DBB_1073, in2 := 7)
   END_RUNG wire#w4
   RUNG wire#w5
      Contact( "DB8000_PART_STATUS".UNIT_2.STATION_1.PART_A.STATUS.MASTER_PART )
   END_RUNG wire#w4
   RUNG wire#w6
      Contact( "U02_TURCK_LD_PART_I" )
   END_RUNG wire#w7
   RUNG wire#w4
      Contact( "DB2031_CYCLES_GENERAL".DRY_CYCLE.CYCLE_SELECTED )
      I_Contact( "DB2031_CYCLES_GENERAL".ROBOT_DRY_CYCLE.CYCLE_SELECTED )
      I_Contact( "DB2031_CYCLES_GENERAL".MANUAL_LOAD_CYCLE.CYCLE_SELECTED )
   END_RUNG wire#w7
   RUNG wire#w4
      Contact( "DB7300_INTERLOCK_GENERAL".LOAD_UNLOAD.UNIT_2.FROM_ROBOT_CELL.PART_LOADED )
   END_RUNG wire#w7
   RUNG wire#w1
      Contact( "DB1101_MACHINE_SEQUENCE".SKIP_FIXTURE_UNIT_02 )
   END_RUNG wire#w7
   RUNG wire#w1
      Contact( "DB2031_CYCLES_GENERAL".RUN_OUT_UNIT_2.CYCLE_SELECTED )
      wire#w8
      Contact( "DB2440_GLOBAL_DATA".GLOBAL_DATA.U02_RN_CYCLE_PART_TYPE )
      Contact( "DB5000_FIX_TABLE_POSITIONS".UNIT_2.FIXTURE_1_OR_3_IN_STA_1 )
      Contact( "DB2031_CYCLES_GENERAL".MANUAL_LOAD_CYCLE.CYCLE_SELECTED )
      Contact( "DB8100_MANUAL_LOADING_PART_STATUS".UNIT_02_NO_FACE_R_PARTS_TO_DELIVER )
   END_RUNG wire#w7
   RUNG wire#w1
      Contact( "DB2031_CYCLES_GENERAL".RUN_OUT_UNIT_2.CYCLE_SELECTED_AUX )
   END_RUNG wire#w8
   RUNG wire#w8
      Contact( "DB2440_GLOBAL_DATA".GLOBAL_DATA.U02_NR_CYCLE_PART_TYPE )
      Contact( "DB5000_FIX_TABLE_POSITIONS".UNIT_2.FIXTURE_2_OR_4_IN_STA_1 )
      Contact( "DB2031_CYCLES_GENERAL".MANUAL_LOAD_CYCLE.CYCLE_SELECTED )
      Contact( "DB8100_MANUAL_LOADING_PART_STATUS".UNIT_02_NO_FACE_N_PARTS_TO_DELIVER )
   END_RUNG wire#w7
   RUNG wire#w1
      I_Contact( "DB2031_CYCLES_GENERAL".MANUAL_LOAD_CYCLE.CYCLE_SELECTED )
      Contact( "DB440_MACHINE_ALARM_DECODING".ALARMS_UNIT_2.GLOBAL.SEOC_ALARMS )
      Contact( "DB7300_INTERLOCK_GENERAL".GENERAL_MACHINE.FROM_ROBOT_TO_UNIT_2.OUT_OF_COLLISION_MACHINE )
   END_RUNG wire#w7
   // the same network as SCL:
   "DB356_M_UNIT_2_STA_0".M_CODES_UNIT_2_STA_0.Ack_M50 := "DB356_M_UNIT_2_STA_0".M_CODES_UNIT_2_STA_0.M50 AND (("DB8000_PART_STATUS".UNIT_2.STATION_1.PART_A.STATUS.PRESENT AND (("DB5000_FIX_TABLE_POSITIONS".UNIT_2.FIXTURE_1_OR_3_IN_STA_1 AND (("DB2440_GLOBAL_DATA".GLOBAL_DATA.U02_RN_CYCLE_PART_TYPE AND "DB8000_PART_STATUS".UNIT_2.STATION_1.PART_A.STATUS.CELL_STATUS.U1_DONE_IN_TRANSIT AND ("DB2401_DBB_DEFINE".PART_STATUS.DBB_1073 = 7)) OR ("DB2440_GLOBAL_DATA".GLOBAL_DATA.U02_NR_CYCLE_PART_TYPE AND "DB8000_PART_STATUS".UNIT_2.STATION_1.PART_A.STATUS.CELL_STATUS.U2_ONE_FACE_DONE_ROTATED AND ("DB2401_DBB_DEFINE".PART_STATUS.DBB_1073 = 11)) OR "DB8000_PART_STATUS".UNIT_2.STATION_1.PART_A.STATUS.MASTER_PART)) OR ("DB5000_FIX_TABLE_POSITIONS".UNIT_2.FIXTURE_2_OR_4_IN_STA_1 AND (("DB2440_GLOBAL_DATA".GLOBAL_DATA.U02_RN_CYCLE_PART_TYPE AND "DB8000_PART_STATUS".UNIT_2.STATION_1.PART_A.STATUS.CELL_STATUS.U2_ONE_FACE_DONE_ROTATED AND ("DB2401_DBB_DEFINE".PART_STATUS.DBB_1073 = 11)) OR ("DB2440_GLOBAL_DATA".GLOBAL_DATA.U02_NR_CYCLE_PART_TYPE AND "DB8000_PART_STATUS".UNIT_2.STATION_1.PART_A.STATUS.CELL_STATUS.U1_DONE_IN_TRANSIT AND ("DB2401_DBB_DEFINE".PART_STATUS.DBB_1073 = 7)) OR "DB8000_PART_STATUS".UNIT_2.STATION_1.PART_A.STATUS.MASTER_PART))) AND (("DB2031_CYCLES_GENERAL".MANUAL_LOAD_CYCLE.CYCLE_SELECTED AND ("DB8100_MANUAL_LOADING_PART_STATUS".UNIT_02_ADD_PART_HMI_BUTTON OR "U02_TURCK_LD_PART_I")) OR ("DB2031_CYCLES_GENERAL".DRY_CYCLE.CYCLE_SELECTED AND NOT "DB2031_CYCLES_GENERAL".ROBOT_DRY_CYCLE.CYCLE_SELECTED AND NOT "DB2031_CYCLES_GENERAL".MANUAL_LOAD_CYCLE.CYCLE_SELECTED) OR "DB7300_INTERLOCK_GENERAL".LOAD_UNLOAD.UNIT_2.FROM_ROBOT_CELL.PART_LOADED)) OR "DB1101_MACHINE_SEQUENCE".SKIP_FIXTURE_UNIT_02 OR (("DB2031_CYCLES_GENERAL".RUN_OUT_UNIT_2.CYCLE_SELECTED OR "DB2031_CYCLES_GENERAL".RUN_OUT_UNIT_2.CYCLE_SELECTED_AUX) AND (("DB2440_GLOBAL_DATA".GLOBAL_DATA.U02_RN_CYCLE_PART_TYPE AND "DB5000_FIX_TABLE_POSITIONS".UNIT_2.FIXTURE_1_OR_3_IN_STA_1 AND "DB2031_CYCLES_GENERAL".MANUAL_LOAD_CYCLE.CYCLE_SELECTED AND "DB8100_MANUAL_LOADING_PART_STATUS".UNIT_02_NO_FACE_R_PARTS_TO_DELIVER) OR ("DB2440_GLOBAL_DATA".GLOBAL_DATA.U02_NR_CYCLE_PART_TYPE AND "DB5000_FIX_TABLE_POSITIONS".UNIT_2.FIXTURE_2_OR_4_IN_STA_1 AND "DB2031_CYCLES_GENERAL".MANUAL_LOAD_CYCLE.CYCLE_SELECTED AND "DB8100_MANUAL_LOADING_PART_STATUS".UNIT_02_NO_FACE_N_PARTS_TO_DELIVER))) OR (NOT "DB2031_CYCLES_GENERAL".MANUAL_LOAD_CYCLE.CYCLE_SELECTED AND "DB440_MACHINE_ALARM_DECODING".ALARMS_UNIT_2.GLOBAL.SEOC_ALARMS AND "DB7300_INTERLOCK_GENERAL".GENERAL_MACHINE.FROM_ROBOT_TO_UNIT_2.OUT_OF_COLLISION_MACHINE));
END_REGION

REGION Network 42: M50-LOAD PART FROM ROBOT (READ IN DISABLE)
   RUNG wire#powerrail
      Contact( "LBP_Chan4".MDyn[50] )
      wire#w1
      I_Contact( "DB356_M_UNIT_2_STA_0".M_CODES_UNIT_2_STA_0.Ack_M50 )
      I_Contact( "DB2120_MPP_ITC_IPC".RESET_FAULTS )
      I_Contact( "DB356_M_UNIT_2_STA_0".M_CODES_UNIT_2_STA_0.M_RESET_PULSE )
      Coil( "DB356_M_UNIT_2_STA_0".M_CODES_UNIT_2_STA_0.M50 )
   END_RUNG
   RUNG wire#powerrail
      Contact( "DB356_M_UNIT_2_STA_0".M_CODES_UNIT_2_STA_0.M50 )
   END_RUNG wire#w1
   // the same network as SCL:
   "DB356_M_UNIT_2_STA_0".M_CODES_UNIT_2_STA_0.M50 := ("LBP_Chan4".MDyn[50] OR "DB356_M_UNIT_2_STA_0".M_CODES_UNIT_2_STA_0.M50) AND NOT "DB356_M_UNIT_2_STA_0".M_CODES_UNIT_2_STA_0.Ack_M50 AND NOT "DB2120_MPP_ITC_IPC".RESET_FAULTS AND NOT "DB356_M_UNIT_2_STA_0".M_CODES_UNIT_2_STA_0.M_RESET_PULSE;
END_REGION

REGION Network 43: ACKNOWLEDGE M51-UNLOAD PART FROM MACHINE (READ IN DISABLE)
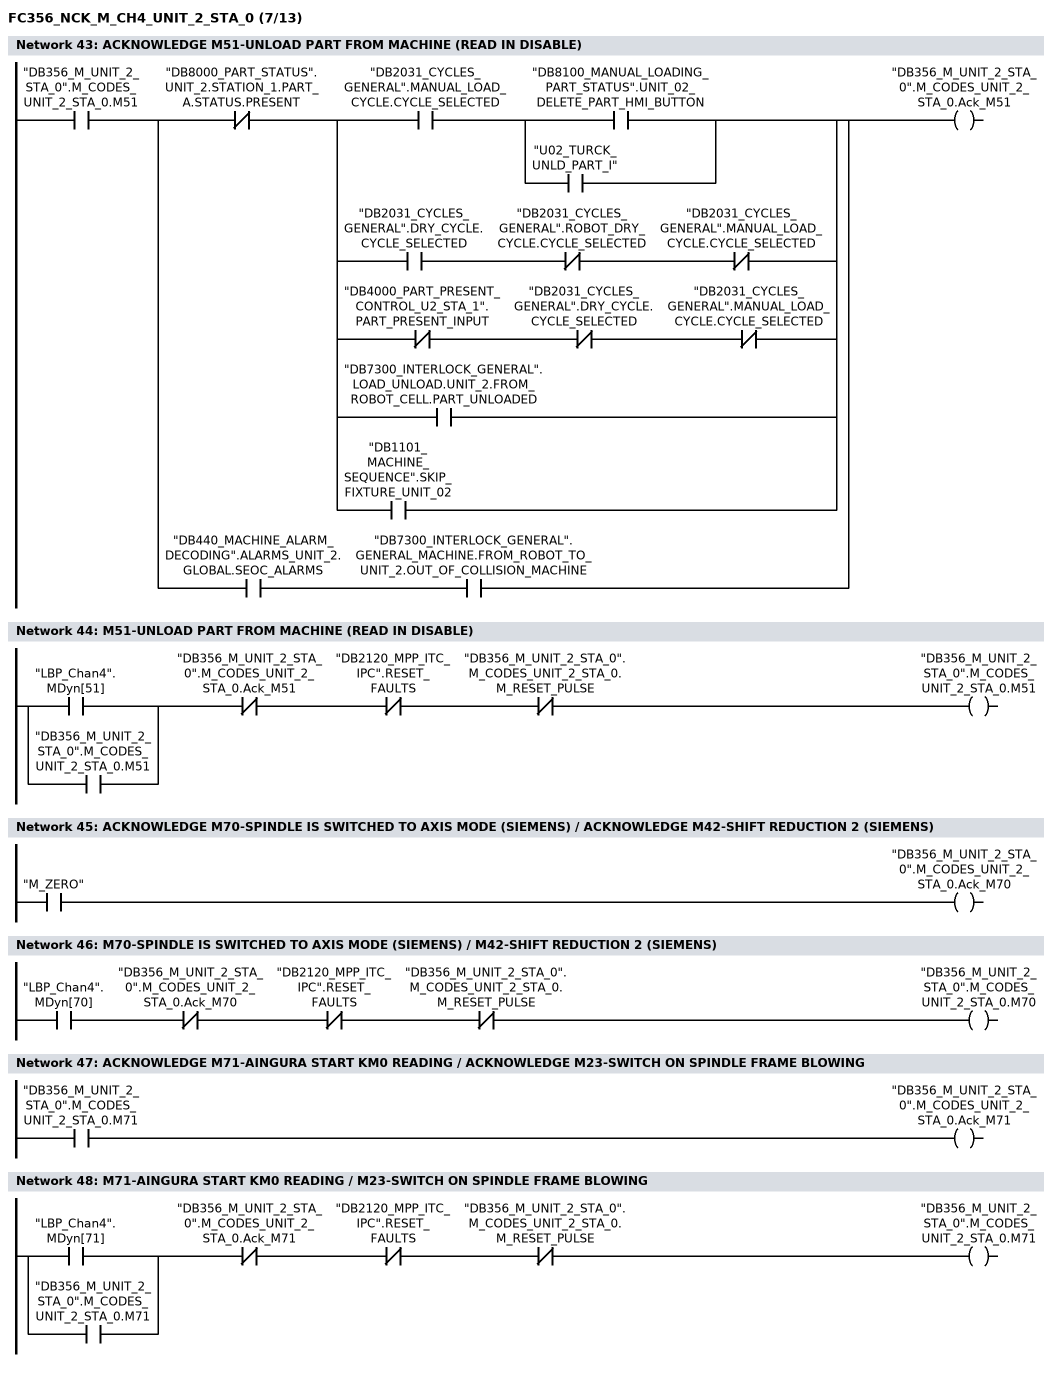
   RUNG wire#powerrail
      Contact( "DB356_M_UNIT_2_STA_0".M_CODES_UNIT_2_STA_0.M51 )
      wire#w1
      I_Contact( "DB8000_PART_STATUS".UNIT_2.STATION_1.PART_A.STATUS.PRESENT )
      wire#w2
      Contact( "DB2031_CYCLES_GENERAL".MANUAL_LOAD_CYCLE.CYCLE_SELECTED )
      wire#w3
      Contact( "DB8100_MANUAL_LOADING_PART_STATUS".UNIT_02_DELETE_PART_HMI_BUTTON )
      wire#w4
      Coil( "DB356_M_UNIT_2_STA_0".M_CODES_UNIT_2_STA_0.Ack_M51 )
   END_RUNG
   RUNG wire#w3
      Contact( "U02_TURCK_UNLD_PART_I" )
   END_RUNG wire#w4
   RUNG wire#w2
      Contact( "DB2031_CYCLES_GENERAL".DRY_CYCLE.CYCLE_SELECTED )
      I_Contact( "DB2031_CYCLES_GENERAL".ROBOT_DRY_CYCLE.CYCLE_SELECTED )
      I_Contact( "DB2031_CYCLES_GENERAL".MANUAL_LOAD_CYCLE.CYCLE_SELECTED )
   END_RUNG wire#w4
   RUNG wire#w2
      I_Contact( "DB4000_PART_PRESENT_CONTROL_U2_STA_1".PART_PRESENT_INPUT )
      I_Contact( "DB2031_CYCLES_GENERAL".DRY_CYCLE.CYCLE_SELECTED )
      I_Contact( "DB2031_CYCLES_GENERAL".MANUAL_LOAD_CYCLE.CYCLE_SELECTED )
   END_RUNG wire#w4
   RUNG wire#w2
      Contact( "DB7300_INTERLOCK_GENERAL".LOAD_UNLOAD.UNIT_2.FROM_ROBOT_CELL.PART_UNLOADED )
   END_RUNG wire#w4
   RUNG wire#w2
      Contact( "DB1101_MACHINE_SEQUENCE".SKIP_FIXTURE_UNIT_02 )
   END_RUNG wire#w4
   RUNG wire#w1
      Contact( "DB440_MACHINE_ALARM_DECODING".ALARMS_UNIT_2.GLOBAL.SEOC_ALARMS )
      Contact( "DB7300_INTERLOCK_GENERAL".GENERAL_MACHINE.FROM_ROBOT_TO_UNIT_2.OUT_OF_COLLISION_MACHINE )
   END_RUNG wire#w4
   // the same network as SCL:
   "DB356_M_UNIT_2_STA_0".M_CODES_UNIT_2_STA_0.Ack_M51 := "DB356_M_UNIT_2_STA_0".M_CODES_UNIT_2_STA_0.M51 AND ((NOT "DB8000_PART_STATUS".UNIT_2.STATION_1.PART_A.STATUS.PRESENT AND (("DB2031_CYCLES_GENERAL".MANUAL_LOAD_CYCLE.CYCLE_SELECTED AND ("DB8100_MANUAL_LOADING_PART_STATUS".UNIT_02_DELETE_PART_HMI_BUTTON OR "U02_TURCK_UNLD_PART_I")) OR ("DB2031_CYCLES_GENERAL".DRY_CYCLE.CYCLE_SELECTED AND NOT "DB2031_CYCLES_GENERAL".ROBOT_DRY_CYCLE.CYCLE_SELECTED AND NOT "DB2031_CYCLES_GENERAL".MANUAL_LOAD_CYCLE.CYCLE_SELECTED) OR (NOT "DB4000_PART_PRESENT_CONTROL_U2_STA_1".PART_PRESENT_INPUT AND NOT "DB2031_CYCLES_GENERAL".DRY_CYCLE.CYCLE_SELECTED AND NOT "DB2031_CYCLES_GENERAL".MANUAL_LOAD_CYCLE.CYCLE_SELECTED) OR "DB7300_INTERLOCK_GENERAL".LOAD_UNLOAD.UNIT_2.FROM_ROBOT_CELL.PART_UNLOADED OR "DB1101_MACHINE_SEQUENCE".SKIP_FIXTURE_UNIT_02)) OR ("DB440_MACHINE_ALARM_DECODING".ALARMS_UNIT_2.GLOBAL.SEOC_ALARMS AND "DB7300_INTERLOCK_GENERAL".GENERAL_MACHINE.FROM_ROBOT_TO_UNIT_2.OUT_OF_COLLISION_MACHINE));
END_REGION

REGION Network 44: M51-UNLOAD PART FROM MACHINE (READ IN DISABLE)
   RUNG wire#powerrail
      Contact( "LBP_Chan4".MDyn[51] )
      wire#w1
      I_Contact( "DB356_M_UNIT_2_STA_0".M_CODES_UNIT_2_STA_0.Ack_M51 )
      I_Contact( "DB2120_MPP_ITC_IPC".RESET_FAULTS )
      I_Contact( "DB356_M_UNIT_2_STA_0".M_CODES_UNIT_2_STA_0.M_RESET_PULSE )
      Coil( "DB356_M_UNIT_2_STA_0".M_CODES_UNIT_2_STA_0.M51 )
   END_RUNG
   RUNG wire#powerrail
      Contact( "DB356_M_UNIT_2_STA_0".M_CODES_UNIT_2_STA_0.M51 )
   END_RUNG wire#w1
   // the same network as SCL:
   "DB356_M_UNIT_2_STA_0".M_CODES_UNIT_2_STA_0.M51 := ("LBP_Chan4".MDyn[51] OR "DB356_M_UNIT_2_STA_0".M_CODES_UNIT_2_STA_0.M51) AND NOT "DB356_M_UNIT_2_STA_0".M_CODES_UNIT_2_STA_0.Ack_M51 AND NOT "DB2120_MPP_ITC_IPC".RESET_FAULTS AND NOT "DB356_M_UNIT_2_STA_0".M_CODES_UNIT_2_STA_0.M_RESET_PULSE;
END_REGION

REGION Network 45: ACKNOWLEDGE M70-SPINDLE IS SWITCHED TO AXIS MODE (SIEMENS) / ACKNOWLEDGE M42-SHIFT REDUCTION 2 (SIEMENS)
   RUNG wire#powerrail
      Contact( "M_ZERO" )
      Coil( "DB356_M_UNIT_2_STA_0".M_CODES_UNIT_2_STA_0.Ack_M70 )
   END_RUNG
   // the same network as SCL:
   "DB356_M_UNIT_2_STA_0".M_CODES_UNIT_2_STA_0.Ack_M70 := "M_ZERO";
END_REGION

REGION Network 46: M70-SPINDLE IS SWITCHED TO AXIS MODE (SIEMENS) / M42-SHIFT REDUCTION 2 (SIEMENS)
   RUNG wire#powerrail
      Contact( "LBP_Chan4".MDyn[70] )
      I_Contact( "DB356_M_UNIT_2_STA_0".M_CODES_UNIT_2_STA_0.Ack_M70 )
      I_Contact( "DB2120_MPP_ITC_IPC".RESET_FAULTS )
      I_Contact( "DB356_M_UNIT_2_STA_0".M_CODES_UNIT_2_STA_0.M_RESET_PULSE )
      Coil( "DB356_M_UNIT_2_STA_0".M_CODES_UNIT_2_STA_0.M70 )
   END_RUNG
   // the same network as SCL:
   "DB356_M_UNIT_2_STA_0".M_CODES_UNIT_2_STA_0.M70 := "LBP_Chan4".MDyn[70] AND NOT "DB356_M_UNIT_2_STA_0".M_CODES_UNIT_2_STA_0.Ack_M70 AND NOT "DB2120_MPP_ITC_IPC".RESET_FAULTS AND NOT "DB356_M_UNIT_2_STA_0".M_CODES_UNIT_2_STA_0.M_RESET_PULSE;
END_REGION

REGION Network 47: ACKNOWLEDGE M71-AINGURA START KM0 READING / ACKNOWLEDGE M23-SWITCH ON SPINDLE FRAME BLOWING
   RUNG wire#powerrail
      Contact( "DB356_M_UNIT_2_STA_0".M_CODES_UNIT_2_STA_0.M71 )
      Coil( "DB356_M_UNIT_2_STA_0".M_CODES_UNIT_2_STA_0.Ack_M71 )
   END_RUNG
   // the same network as SCL:
   "DB356_M_UNIT_2_STA_0".M_CODES_UNIT_2_STA_0.Ack_M71 := "DB356_M_UNIT_2_STA_0".M_CODES_UNIT_2_STA_0.M71;
END_REGION

REGION Network 48: M71-AINGURA START KM0 READING / M23-SWITCH ON SPINDLE FRAME BLOWING
   RUNG wire#powerrail
      Contact( "LBP_Chan4".MDyn[71] )
      wire#w1
      I_Contact( "DB356_M_UNIT_2_STA_0".M_CODES_UNIT_2_STA_0.Ack_M71 )
      I_Contact( "DB2120_MPP_ITC_IPC".RESET_FAULTS )
      I_Contact( "DB356_M_UNIT_2_STA_0".M_CODES_UNIT_2_STA_0.M_RESET_PULSE )
      Coil( "DB356_M_UNIT_2_STA_0".M_CODES_UNIT_2_STA_0.M71 )
   END_RUNG
   RUNG wire#powerrail
      Contact( "DB356_M_UNIT_2_STA_0".M_CODES_UNIT_2_STA_0.M71 )
   END_RUNG wire#w1
   // the same network as SCL:
   "DB356_M_UNIT_2_STA_0".M_CODES_UNIT_2_STA_0.M71 := ("LBP_Chan4".MDyn[71] OR "DB356_M_UNIT_2_STA_0".M_CODES_UNIT_2_STA_0.M71) AND NOT "DB356_M_UNIT_2_STA_0".M_CODES_UNIT_2_STA_0.Ack_M71 AND NOT "DB2120_MPP_ITC_IPC".RESET_FAULTS AND NOT "DB356_M_UNIT_2_STA_0".M_CODES_UNIT_2_STA_0.M_RESET_PULSE;
END_REGION

REGION Network 49: ACKNOWLEDGE M72-AINGURA STOP KM0 READING / ACKNOWLEDGE M23-SWITCH ON SPINDLE FRAME BLOWING
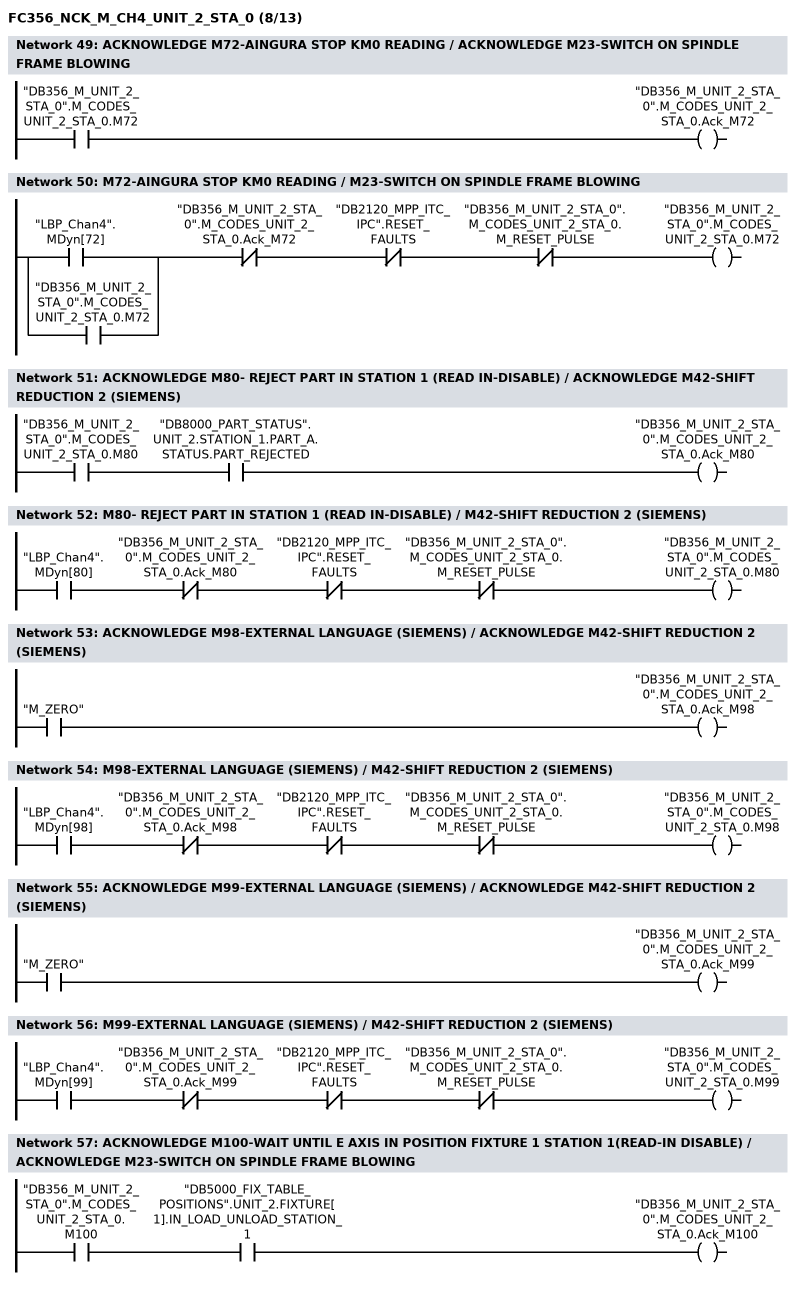
   RUNG wire#powerrail
      Contact( "DB356_M_UNIT_2_STA_0".M_CODES_UNIT_2_STA_0.M72 )
      Coil( "DB356_M_UNIT_2_STA_0".M_CODES_UNIT_2_STA_0.Ack_M72 )
   END_RUNG
   // the same network as SCL:
   "DB356_M_UNIT_2_STA_0".M_CODES_UNIT_2_STA_0.Ack_M72 := "DB356_M_UNIT_2_STA_0".M_CODES_UNIT_2_STA_0.M72;
END_REGION

REGION Network 50: M72-AINGURA STOP KM0 READING / M23-SWITCH ON SPINDLE FRAME BLOWING
   RUNG wire#powerrail
      Contact( "LBP_Chan4".MDyn[72] )
      wire#w1
      I_Contact( "DB356_M_UNIT_2_STA_0".M_CODES_UNIT_2_STA_0.Ack_M72 )
      I_Contact( "DB2120_MPP_ITC_IPC".RESET_FAULTS )
      I_Contact( "DB356_M_UNIT_2_STA_0".M_CODES_UNIT_2_STA_0.M_RESET_PULSE )
      Coil( "DB356_M_UNIT_2_STA_0".M_CODES_UNIT_2_STA_0.M72 )
   END_RUNG
   RUNG wire#powerrail
      Contact( "DB356_M_UNIT_2_STA_0".M_CODES_UNIT_2_STA_0.M72 )
   END_RUNG wire#w1
   // the same network as SCL:
   "DB356_M_UNIT_2_STA_0".M_CODES_UNIT_2_STA_0.M72 := ("LBP_Chan4".MDyn[72] OR "DB356_M_UNIT_2_STA_0".M_CODES_UNIT_2_STA_0.M72) AND NOT "DB356_M_UNIT_2_STA_0".M_CODES_UNIT_2_STA_0.Ack_M72 AND NOT "DB2120_MPP_ITC_IPC".RESET_FAULTS AND NOT "DB356_M_UNIT_2_STA_0".M_CODES_UNIT_2_STA_0.M_RESET_PULSE;
END_REGION

REGION Network 51: ACKNOWLEDGE M80- REJECT PART IN STATION 1 (READ IN-DISABLE) / ACKNOWLEDGE M42-SHIFT REDUCTION 2 (SIEMENS)
   RUNG wire#powerrail
      Contact( "DB356_M_UNIT_2_STA_0".M_CODES_UNIT_2_STA_0.M80 )
      Contact( "DB8000_PART_STATUS".UNIT_2.STATION_1.PART_A.STATUS.PART_REJECTED )
      Coil( "DB356_M_UNIT_2_STA_0".M_CODES_UNIT_2_STA_0.Ack_M80 )
   END_RUNG
   // the same network as SCL:
   "DB356_M_UNIT_2_STA_0".M_CODES_UNIT_2_STA_0.Ack_M80 := "DB356_M_UNIT_2_STA_0".M_CODES_UNIT_2_STA_0.M80 AND "DB8000_PART_STATUS".UNIT_2.STATION_1.PART_A.STATUS.PART_REJECTED;
END_REGION

REGION Network 52: M80- REJECT PART IN STATION 1 (READ IN-DISABLE) / M42-SHIFT REDUCTION 2 (SIEMENS)
   RUNG wire#powerrail
      Contact( "LBP_Chan4".MDyn[80] )
      I_Contact( "DB356_M_UNIT_2_STA_0".M_CODES_UNIT_2_STA_0.Ack_M80 )
      I_Contact( "DB2120_MPP_ITC_IPC".RESET_FAULTS )
      I_Contact( "DB356_M_UNIT_2_STA_0".M_CODES_UNIT_2_STA_0.M_RESET_PULSE )
      Coil( "DB356_M_UNIT_2_STA_0".M_CODES_UNIT_2_STA_0.M80 )
   END_RUNG
   // the same network as SCL:
   "DB356_M_UNIT_2_STA_0".M_CODES_UNIT_2_STA_0.M80 := "LBP_Chan4".MDyn[80] AND NOT "DB356_M_UNIT_2_STA_0".M_CODES_UNIT_2_STA_0.Ack_M80 AND NOT "DB2120_MPP_ITC_IPC".RESET_FAULTS AND NOT "DB356_M_UNIT_2_STA_0".M_CODES_UNIT_2_STA_0.M_RESET_PULSE;
END_REGION

REGION Network 53: ACKNOWLEDGE M98-EXTERNAL LANGUAGE (SIEMENS) / ACKNOWLEDGE M42-SHIFT REDUCTION 2 (SIEMENS)
   RUNG wire#powerrail
      Contact( "M_ZERO" )
      Coil( "DB356_M_UNIT_2_STA_0".M_CODES_UNIT_2_STA_0.Ack_M98 )
   END_RUNG
   // the same network as SCL:
   "DB356_M_UNIT_2_STA_0".M_CODES_UNIT_2_STA_0.Ack_M98 := "M_ZERO";
END_REGION

REGION Network 54: M98-EXTERNAL LANGUAGE (SIEMENS) / M42-SHIFT REDUCTION 2 (SIEMENS)
   RUNG wire#powerrail
      Contact( "LBP_Chan4".MDyn[98] )
      I_Contact( "DB356_M_UNIT_2_STA_0".M_CODES_UNIT_2_STA_0.Ack_M98 )
      I_Contact( "DB2120_MPP_ITC_IPC".RESET_FAULTS )
      I_Contact( "DB356_M_UNIT_2_STA_0".M_CODES_UNIT_2_STA_0.M_RESET_PULSE )
      Coil( "DB356_M_UNIT_2_STA_0".M_CODES_UNIT_2_STA_0.M98 )
   END_RUNG
   // the same network as SCL:
   "DB356_M_UNIT_2_STA_0".M_CODES_UNIT_2_STA_0.M98 := "LBP_Chan4".MDyn[98] AND NOT "DB356_M_UNIT_2_STA_0".M_CODES_UNIT_2_STA_0.Ack_M98 AND NOT "DB2120_MPP_ITC_IPC".RESET_FAULTS AND NOT "DB356_M_UNIT_2_STA_0".M_CODES_UNIT_2_STA_0.M_RESET_PULSE;
END_REGION

REGION Network 55: ACKNOWLEDGE M99-EXTERNAL LANGUAGE (SIEMENS) / ACKNOWLEDGE M42-SHIFT REDUCTION 2 (SIEMENS)
   RUNG wire#powerrail
      Contact( "M_ZERO" )
      Coil( "DB356_M_UNIT_2_STA_0".M_CODES_UNIT_2_STA_0.Ack_M99 )
   END_RUNG
   // the same network as SCL:
   "DB356_M_UNIT_2_STA_0".M_CODES_UNIT_2_STA_0.Ack_M99 := "M_ZERO";
END_REGION

REGION Network 56: M99-EXTERNAL LANGUAGE (SIEMENS) / M42-SHIFT REDUCTION 2 (SIEMENS)
   RUNG wire#powerrail
      Contact( "LBP_Chan4".MDyn[99] )
      I_Contact( "DB356_M_UNIT_2_STA_0".M_CODES_UNIT_2_STA_0.Ack_M99 )
      I_Contact( "DB2120_MPP_ITC_IPC".RESET_FAULTS )
      I_Contact( "DB356_M_UNIT_2_STA_0".M_CODES_UNIT_2_STA_0.M_RESET_PULSE )
      Coil( "DB356_M_UNIT_2_STA_0".M_CODES_UNIT_2_STA_0.M99 )
   END_RUNG
   // the same network as SCL:
   "DB356_M_UNIT_2_STA_0".M_CODES_UNIT_2_STA_0.M99 := "LBP_Chan4".MDyn[99] AND NOT "DB356_M_UNIT_2_STA_0".M_CODES_UNIT_2_STA_0.Ack_M99 AND NOT "DB2120_MPP_ITC_IPC".RESET_FAULTS AND NOT "DB356_M_UNIT_2_STA_0".M_CODES_UNIT_2_STA_0.M_RESET_PULSE;
END_REGION

REGION Network 57: ACKNOWLEDGE M100-WAIT UNTIL E AXIS IN POSITION FIXTURE 1 STATION 1(READ-IN DISABLE) / ACKNOWLEDGE M23-SWITCH ON SPINDLE FRAME BLOWING
   RUNG wire#powerrail
      Contact( "DB356_M_UNIT_2_STA_0".M_CODES_UNIT_2_STA_0.M100 )
      Contact( "DB5000_FIX_TABLE_POSITIONS".UNIT_2.FIXTURE[1].IN_LOAD_UNLOAD_STATION_1 )
      Coil( "DB356_M_UNIT_2_STA_0".M_CODES_UNIT_2_STA_0.Ack_M100 )
   END_RUNG
   // the same network as SCL:
   "DB356_M_UNIT_2_STA_0".M_CODES_UNIT_2_STA_0.Ack_M100 := "DB356_M_UNIT_2_STA_0".M_CODES_UNIT_2_STA_0.M100 AND "DB5000_FIX_TABLE_POSITIONS".UNIT_2.FIXTURE[1].IN_LOAD_UNLOAD_STATION_1;
END_REGION

REGION Network 58: M100-WAIT UNTIL E AXIS IN POSITION FIXTURE 1 STATION 1(READ-IN DISABLE) / M23-SWITCH ON SPINDLE FRAME BLOWING
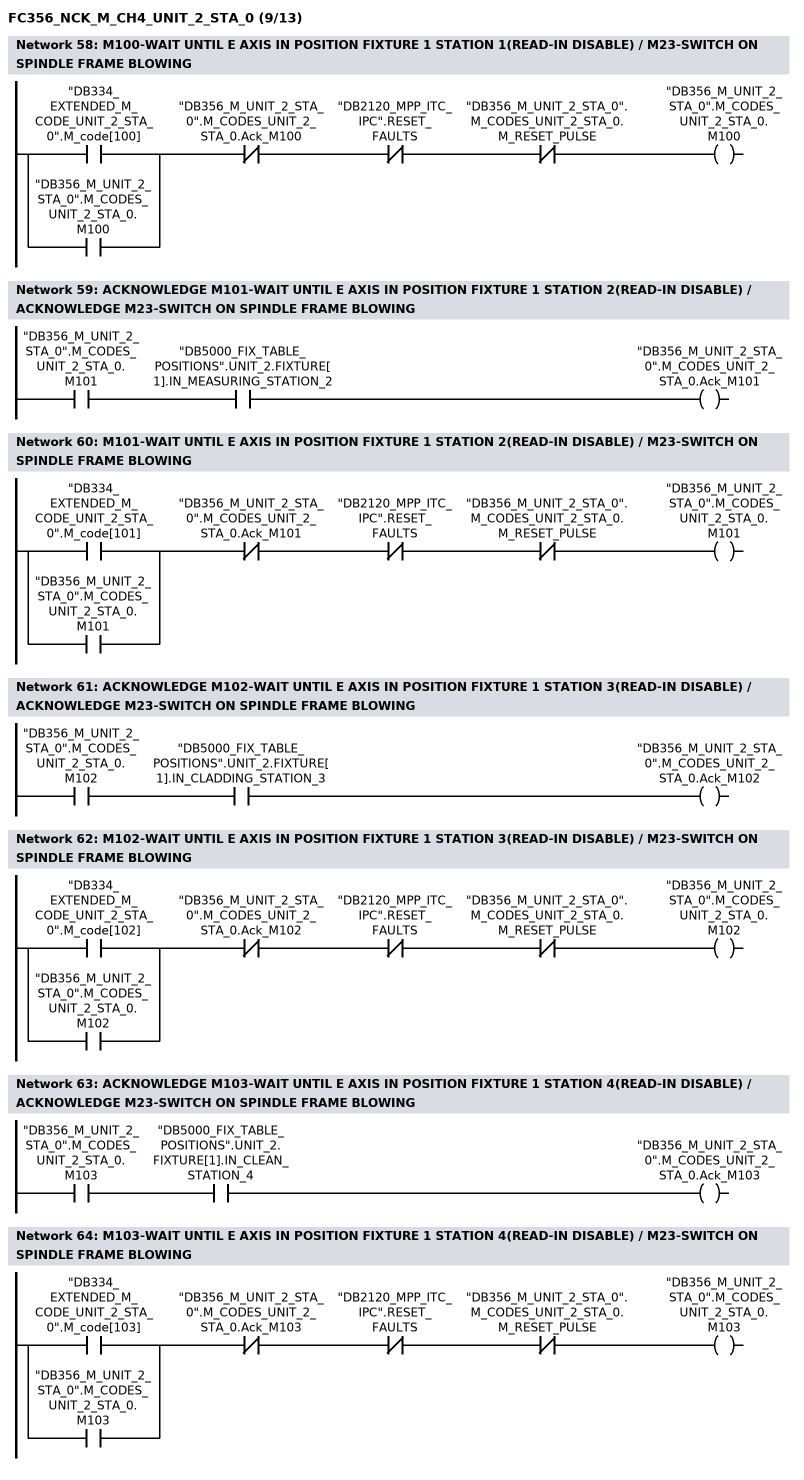
   RUNG wire#powerrail
      Contact( "DB334_EXTENDED_M_CODE_UNIT_2_STA_0".M_code[100] )
      wire#w1
      I_Contact( "DB356_M_UNIT_2_STA_0".M_CODES_UNIT_2_STA_0.Ack_M100 )
      I_Contact( "DB2120_MPP_ITC_IPC".RESET_FAULTS )
      I_Contact( "DB356_M_UNIT_2_STA_0".M_CODES_UNIT_2_STA_0.M_RESET_PULSE )
      Coil( "DB356_M_UNIT_2_STA_0".M_CODES_UNIT_2_STA_0.M100 )
   END_RUNG
   RUNG wire#powerrail
      Contact( "DB356_M_UNIT_2_STA_0".M_CODES_UNIT_2_STA_0.M100 )
   END_RUNG wire#w1
   // the same network as SCL:
   "DB356_M_UNIT_2_STA_0".M_CODES_UNIT_2_STA_0.M100 := ("DB334_EXTENDED_M_CODE_UNIT_2_STA_0".M_code[100] OR "DB356_M_UNIT_2_STA_0".M_CODES_UNIT_2_STA_0.M100) AND NOT "DB356_M_UNIT_2_STA_0".M_CODES_UNIT_2_STA_0.Ack_M100 AND NOT "DB2120_MPP_ITC_IPC".RESET_FAULTS AND NOT "DB356_M_UNIT_2_STA_0".M_CODES_UNIT_2_STA_0.M_RESET_PULSE;
END_REGION

REGION Network 59: ACKNOWLEDGE M101-WAIT UNTIL E AXIS IN POSITION FIXTURE 1 STATION 2(READ-IN DISABLE) / ACKNOWLEDGE M23-SWITCH ON SPINDLE FRAME BLOWING
   RUNG wire#powerrail
      Contact( "DB356_M_UNIT_2_STA_0".M_CODES_UNIT_2_STA_0.M101 )
      Contact( "DB5000_FIX_TABLE_POSITIONS".UNIT_2.FIXTURE[1].IN_MEASURING_STATION_2 )
      Coil( "DB356_M_UNIT_2_STA_0".M_CODES_UNIT_2_STA_0.Ack_M101 )
   END_RUNG
   // the same network as SCL:
   "DB356_M_UNIT_2_STA_0".M_CODES_UNIT_2_STA_0.Ack_M101 := "DB356_M_UNIT_2_STA_0".M_CODES_UNIT_2_STA_0.M101 AND "DB5000_FIX_TABLE_POSITIONS".UNIT_2.FIXTURE[1].IN_MEASURING_STATION_2;
END_REGION

REGION Network 60: M101-WAIT UNTIL E AXIS IN POSITION FIXTURE 1 STATION 2(READ-IN DISABLE) / M23-SWITCH ON SPINDLE FRAME BLOWING
   RUNG wire#powerrail
      Contact( "DB334_EXTENDED_M_CODE_UNIT_2_STA_0".M_code[101] )
      wire#w1
      I_Contact( "DB356_M_UNIT_2_STA_0".M_CODES_UNIT_2_STA_0.Ack_M101 )
      I_Contact( "DB2120_MPP_ITC_IPC".RESET_FAULTS )
      I_Contact( "DB356_M_UNIT_2_STA_0".M_CODES_UNIT_2_STA_0.M_RESET_PULSE )
      Coil( "DB356_M_UNIT_2_STA_0".M_CODES_UNIT_2_STA_0.M101 )
   END_RUNG
   RUNG wire#powerrail
      Contact( "DB356_M_UNIT_2_STA_0".M_CODES_UNIT_2_STA_0.M101 )
   END_RUNG wire#w1
   // the same network as SCL:
   "DB356_M_UNIT_2_STA_0".M_CODES_UNIT_2_STA_0.M101 := ("DB334_EXTENDED_M_CODE_UNIT_2_STA_0".M_code[101] OR "DB356_M_UNIT_2_STA_0".M_CODES_UNIT_2_STA_0.M101) AND NOT "DB356_M_UNIT_2_STA_0".M_CODES_UNIT_2_STA_0.Ack_M101 AND NOT "DB2120_MPP_ITC_IPC".RESET_FAULTS AND NOT "DB356_M_UNIT_2_STA_0".M_CODES_UNIT_2_STA_0.M_RESET_PULSE;
END_REGION

REGION Network 61: ACKNOWLEDGE M102-WAIT UNTIL E AXIS IN POSITION FIXTURE 1 STATION 3(READ-IN DISABLE) / ACKNOWLEDGE M23-SWITCH ON SPINDLE FRAME BLOWING
   RUNG wire#powerrail
      Contact( "DB356_M_UNIT_2_STA_0".M_CODES_UNIT_2_STA_0.M102 )
      Contact( "DB5000_FIX_TABLE_POSITIONS".UNIT_2.FIXTURE[1].IN_CLADDING_STATION_3 )
      Coil( "DB356_M_UNIT_2_STA_0".M_CODES_UNIT_2_STA_0.Ack_M102 )
   END_RUNG
   // the same network as SCL:
   "DB356_M_UNIT_2_STA_0".M_CODES_UNIT_2_STA_0.Ack_M102 := "DB356_M_UNIT_2_STA_0".M_CODES_UNIT_2_STA_0.M102 AND "DB5000_FIX_TABLE_POSITIONS".UNIT_2.FIXTURE[1].IN_CLADDING_STATION_3;
END_REGION

REGION Network 62: M102-WAIT UNTIL E AXIS IN POSITION FIXTURE 1 STATION 3(READ-IN DISABLE) / M23-SWITCH ON SPINDLE FRAME BLOWING
   RUNG wire#powerrail
      Contact( "DB334_EXTENDED_M_CODE_UNIT_2_STA_0".M_code[102] )
      wire#w1
      I_Contact( "DB356_M_UNIT_2_STA_0".M_CODES_UNIT_2_STA_0.Ack_M102 )
      I_Contact( "DB2120_MPP_ITC_IPC".RESET_FAULTS )
      I_Contact( "DB356_M_UNIT_2_STA_0".M_CODES_UNIT_2_STA_0.M_RESET_PULSE )
      Coil( "DB356_M_UNIT_2_STA_0".M_CODES_UNIT_2_STA_0.M102 )
   END_RUNG
   RUNG wire#powerrail
      Contact( "DB356_M_UNIT_2_STA_0".M_CODES_UNIT_2_STA_0.M102 )
   END_RUNG wire#w1
   // the same network as SCL:
   "DB356_M_UNIT_2_STA_0".M_CODES_UNIT_2_STA_0.M102 := ("DB334_EXTENDED_M_CODE_UNIT_2_STA_0".M_code[102] OR "DB356_M_UNIT_2_STA_0".M_CODES_UNIT_2_STA_0.M102) AND NOT "DB356_M_UNIT_2_STA_0".M_CODES_UNIT_2_STA_0.Ack_M102 AND NOT "DB2120_MPP_ITC_IPC".RESET_FAULTS AND NOT "DB356_M_UNIT_2_STA_0".M_CODES_UNIT_2_STA_0.M_RESET_PULSE;
END_REGION

REGION Network 63: ACKNOWLEDGE M103-WAIT UNTIL E AXIS IN POSITION FIXTURE 1 STATION 4(READ-IN DISABLE) / ACKNOWLEDGE M23-SWITCH ON SPINDLE FRAME BLOWING
   RUNG wire#powerrail
      Contact( "DB356_M_UNIT_2_STA_0".M_CODES_UNIT_2_STA_0.M103 )
      Contact( "DB5000_FIX_TABLE_POSITIONS".UNIT_2.FIXTURE[1].IN_CLEAN_STATION_4 )
      Coil( "DB356_M_UNIT_2_STA_0".M_CODES_UNIT_2_STA_0.Ack_M103 )
   END_RUNG
   // the same network as SCL:
   "DB356_M_UNIT_2_STA_0".M_CODES_UNIT_2_STA_0.Ack_M103 := "DB356_M_UNIT_2_STA_0".M_CODES_UNIT_2_STA_0.M103 AND "DB5000_FIX_TABLE_POSITIONS".UNIT_2.FIXTURE[1].IN_CLEAN_STATION_4;
END_REGION

REGION Network 64: M103-WAIT UNTIL E AXIS IN POSITION FIXTURE 1 STATION 4(READ-IN DISABLE) / M23-SWITCH ON SPINDLE FRAME BLOWING
   RUNG wire#powerrail
      Contact( "DB334_EXTENDED_M_CODE_UNIT_2_STA_0".M_code[103] )
      wire#w1
      I_Contact( "DB356_M_UNIT_2_STA_0".M_CODES_UNIT_2_STA_0.Ack_M103 )
      I_Contact( "DB2120_MPP_ITC_IPC".RESET_FAULTS )
      I_Contact( "DB356_M_UNIT_2_STA_0".M_CODES_UNIT_2_STA_0.M_RESET_PULSE )
      Coil( "DB356_M_UNIT_2_STA_0".M_CODES_UNIT_2_STA_0.M103 )
   END_RUNG
   RUNG wire#powerrail
      Contact( "DB356_M_UNIT_2_STA_0".M_CODES_UNIT_2_STA_0.M103 )
   END_RUNG wire#w1
   // the same network as SCL:
   "DB356_M_UNIT_2_STA_0".M_CODES_UNIT_2_STA_0.M103 := ("DB334_EXTENDED_M_CODE_UNIT_2_STA_0".M_code[103] OR "DB356_M_UNIT_2_STA_0".M_CODES_UNIT_2_STA_0.M103) AND NOT "DB356_M_UNIT_2_STA_0".M_CODES_UNIT_2_STA_0.Ack_M103 AND NOT "DB2120_MPP_ITC_IPC".RESET_FAULTS AND NOT "DB356_M_UNIT_2_STA_0".M_CODES_UNIT_2_STA_0.M_RESET_PULSE;
END_REGION

REGION Network 65: ACKNOWLEDGE M110-RETURN UP SEALING STRUCTURE (READ IN DISABLE) / ACKNOWLEDGE M32-UNBLOCK TABLE
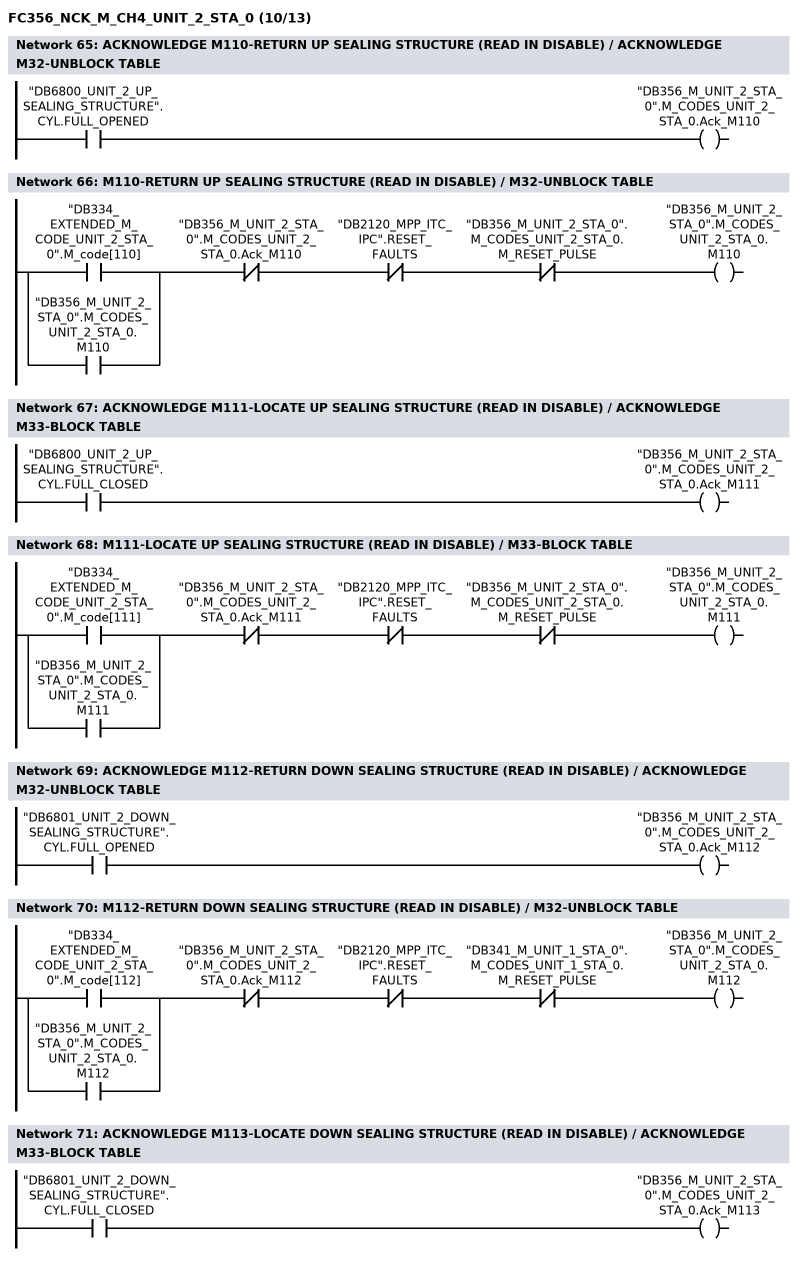
   RUNG wire#powerrail
      Contact( "DB6800_UNIT_2_UP_SEALING_STRUCTURE".CYL.FULL_OPENED )
      Coil( "DB356_M_UNIT_2_STA_0".M_CODES_UNIT_2_STA_0.Ack_M110 )
   END_RUNG
   // the same network as SCL:
   "DB356_M_UNIT_2_STA_0".M_CODES_UNIT_2_STA_0.Ack_M110 := "DB6800_UNIT_2_UP_SEALING_STRUCTURE".CYL.FULL_OPENED;
END_REGION

REGION Network 66: M110-RETURN UP SEALING STRUCTURE (READ IN DISABLE) / M32-UNBLOCK TABLE
   RUNG wire#powerrail
      Contact( "DB334_EXTENDED_M_CODE_UNIT_2_STA_0".M_code[110] )
      wire#w1
      I_Contact( "DB356_M_UNIT_2_STA_0".M_CODES_UNIT_2_STA_0.Ack_M110 )
      I_Contact( "DB2120_MPP_ITC_IPC".RESET_FAULTS )
      I_Contact( "DB356_M_UNIT_2_STA_0".M_CODES_UNIT_2_STA_0.M_RESET_PULSE )
      Coil( "DB356_M_UNIT_2_STA_0".M_CODES_UNIT_2_STA_0.M110 )
   END_RUNG
   RUNG wire#powerrail
      Contact( "DB356_M_UNIT_2_STA_0".M_CODES_UNIT_2_STA_0.M110 )
   END_RUNG wire#w1
   // the same network as SCL:
   "DB356_M_UNIT_2_STA_0".M_CODES_UNIT_2_STA_0.M110 := ("DB334_EXTENDED_M_CODE_UNIT_2_STA_0".M_code[110] OR "DB356_M_UNIT_2_STA_0".M_CODES_UNIT_2_STA_0.M110) AND NOT "DB356_M_UNIT_2_STA_0".M_CODES_UNIT_2_STA_0.Ack_M110 AND NOT "DB2120_MPP_ITC_IPC".RESET_FAULTS AND NOT "DB356_M_UNIT_2_STA_0".M_CODES_UNIT_2_STA_0.M_RESET_PULSE;
END_REGION

REGION Network 67: ACKNOWLEDGE M111-LOCATE UP SEALING STRUCTURE (READ IN DISABLE) / ACKNOWLEDGE M33-BLOCK TABLE
   RUNG wire#powerrail
      Contact( "DB6800_UNIT_2_UP_SEALING_STRUCTURE".CYL.FULL_CLOSED )
      Coil( "DB356_M_UNIT_2_STA_0".M_CODES_UNIT_2_STA_0.Ack_M111 )
   END_RUNG
   // the same network as SCL:
   "DB356_M_UNIT_2_STA_0".M_CODES_UNIT_2_STA_0.Ack_M111 := "DB6800_UNIT_2_UP_SEALING_STRUCTURE".CYL.FULL_CLOSED;
END_REGION

REGION Network 68: M111-LOCATE UP SEALING STRUCTURE (READ IN DISABLE) / M33-BLOCK TABLE
   RUNG wire#powerrail
      Contact( "DB334_EXTENDED_M_CODE_UNIT_2_STA_0".M_code[111] )
      wire#w1
      I_Contact( "DB356_M_UNIT_2_STA_0".M_CODES_UNIT_2_STA_0.Ack_M111 )
      I_Contact( "DB2120_MPP_ITC_IPC".RESET_FAULTS )
      I_Contact( "DB356_M_UNIT_2_STA_0".M_CODES_UNIT_2_STA_0.M_RESET_PULSE )
      Coil( "DB356_M_UNIT_2_STA_0".M_CODES_UNIT_2_STA_0.M111 )
   END_RUNG
   RUNG wire#powerrail
      Contact( "DB356_M_UNIT_2_STA_0".M_CODES_UNIT_2_STA_0.M111 )
   END_RUNG wire#w1
   // the same network as SCL:
   "DB356_M_UNIT_2_STA_0".M_CODES_UNIT_2_STA_0.M111 := ("DB334_EXTENDED_M_CODE_UNIT_2_STA_0".M_code[111] OR "DB356_M_UNIT_2_STA_0".M_CODES_UNIT_2_STA_0.M111) AND NOT "DB356_M_UNIT_2_STA_0".M_CODES_UNIT_2_STA_0.Ack_M111 AND NOT "DB2120_MPP_ITC_IPC".RESET_FAULTS AND NOT "DB356_M_UNIT_2_STA_0".M_CODES_UNIT_2_STA_0.M_RESET_PULSE;
END_REGION

REGION Network 69: ACKNOWLEDGE M112-RETURN DOWN SEALING STRUCTURE (READ IN DISABLE) / ACKNOWLEDGE M32-UNBLOCK TABLE
   RUNG wire#powerrail
      Contact( "DB6801_UNIT_2_DOWN_SEALING_STRUCTURE".CYL.FULL_OPENED )
      Coil( "DB356_M_UNIT_2_STA_0".M_CODES_UNIT_2_STA_0.Ack_M112 )
   END_RUNG
   // the same network as SCL:
   "DB356_M_UNIT_2_STA_0".M_CODES_UNIT_2_STA_0.Ack_M112 := "DB6801_UNIT_2_DOWN_SEALING_STRUCTURE".CYL.FULL_OPENED;
END_REGION

REGION Network 70: M112-RETURN DOWN SEALING STRUCTURE (READ IN DISABLE) / M32-UNBLOCK TABLE
   RUNG wire#powerrail
      Contact( "DB334_EXTENDED_M_CODE_UNIT_2_STA_0".M_code[112] )
      wire#w1
      I_Contact( "DB356_M_UNIT_2_STA_0".M_CODES_UNIT_2_STA_0.Ack_M112 )
      I_Contact( "DB2120_MPP_ITC_IPC".RESET_FAULTS )
      I_Contact( "DB341_M_UNIT_1_STA_0".M_CODES_UNIT_1_STA_0.M_RESET_PULSE )
      Coil( "DB356_M_UNIT_2_STA_0".M_CODES_UNIT_2_STA_0.M112 )
   END_RUNG
   RUNG wire#powerrail
      Contact( "DB356_M_UNIT_2_STA_0".M_CODES_UNIT_2_STA_0.M112 )
   END_RUNG wire#w1
   // the same network as SCL:
   "DB356_M_UNIT_2_STA_0".M_CODES_UNIT_2_STA_0.M112 := ("DB334_EXTENDED_M_CODE_UNIT_2_STA_0".M_code[112] OR "DB356_M_UNIT_2_STA_0".M_CODES_UNIT_2_STA_0.M112) AND NOT "DB356_M_UNIT_2_STA_0".M_CODES_UNIT_2_STA_0.Ack_M112 AND NOT "DB2120_MPP_ITC_IPC".RESET_FAULTS AND NOT "DB341_M_UNIT_1_STA_0".M_CODES_UNIT_1_STA_0.M_RESET_PULSE;
END_REGION

REGION Network 71: ACKNOWLEDGE M113-LOCATE DOWN SEALING STRUCTURE (READ IN DISABLE) / ACKNOWLEDGE M33-BLOCK TABLE
   RUNG wire#powerrail
      Contact( "DB6801_UNIT_2_DOWN_SEALING_STRUCTURE".CYL.FULL_CLOSED )
      Coil( "DB356_M_UNIT_2_STA_0".M_CODES_UNIT_2_STA_0.Ack_M113 )
   END_RUNG
   // the same network as SCL:
   "DB356_M_UNIT_2_STA_0".M_CODES_UNIT_2_STA_0.Ack_M113 := "DB6801_UNIT_2_DOWN_SEALING_STRUCTURE".CYL.FULL_CLOSED;
END_REGION

REGION Network 72: M113-LOCATE DOWN SEALING STRUCTURE (READ IN DISABLE) / M33-BLOCK TABLE
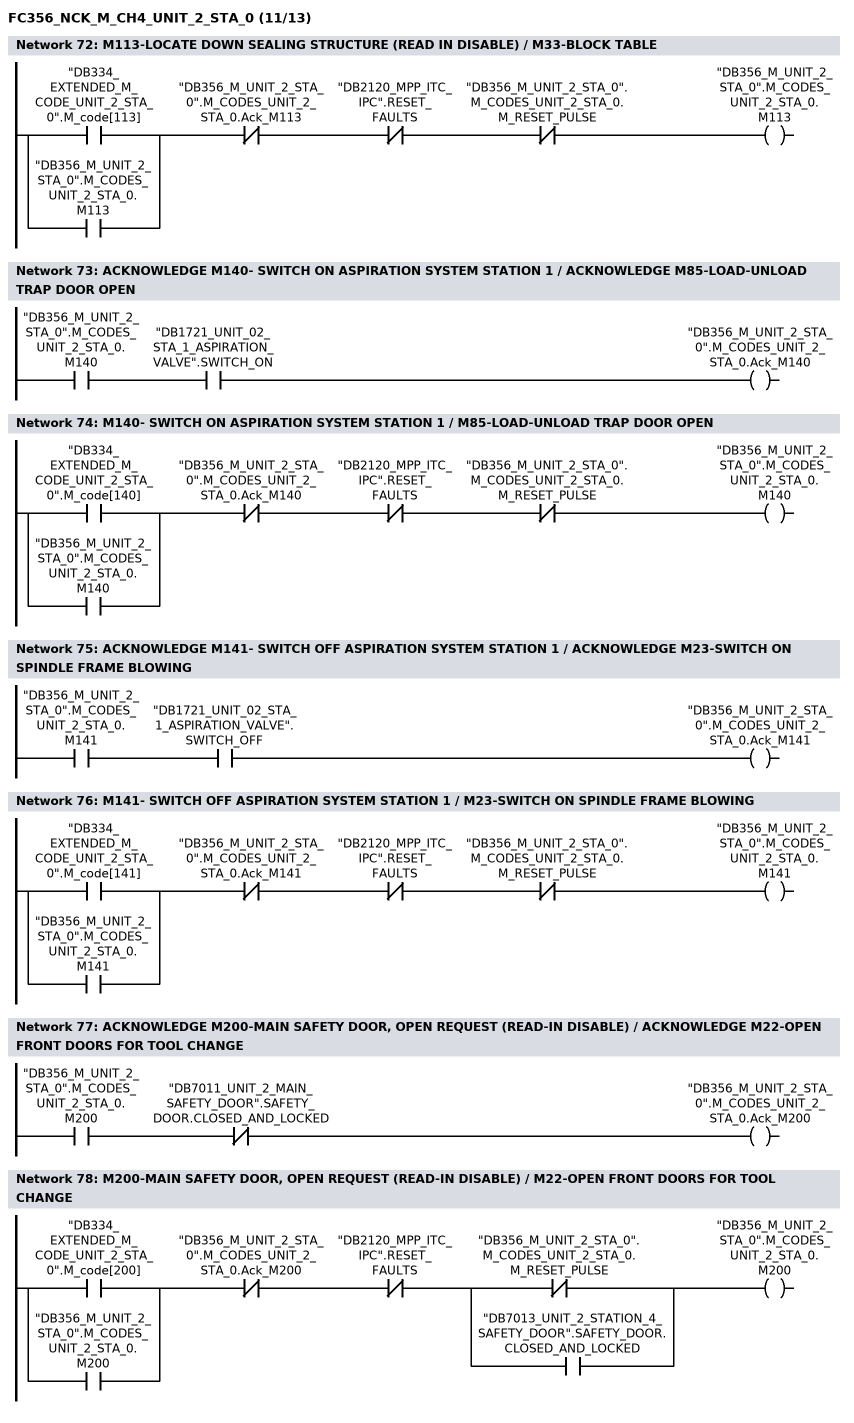
   RUNG wire#powerrail
      Contact( "DB334_EXTENDED_M_CODE_UNIT_2_STA_0".M_code[113] )
      wire#w1
      I_Contact( "DB356_M_UNIT_2_STA_0".M_CODES_UNIT_2_STA_0.Ack_M113 )
      I_Contact( "DB2120_MPP_ITC_IPC".RESET_FAULTS )
      I_Contact( "DB356_M_UNIT_2_STA_0".M_CODES_UNIT_2_STA_0.M_RESET_PULSE )
      Coil( "DB356_M_UNIT_2_STA_0".M_CODES_UNIT_2_STA_0.M113 )
   END_RUNG
   RUNG wire#powerrail
      Contact( "DB356_M_UNIT_2_STA_0".M_CODES_UNIT_2_STA_0.M113 )
   END_RUNG wire#w1
   // the same network as SCL:
   "DB356_M_UNIT_2_STA_0".M_CODES_UNIT_2_STA_0.M113 := ("DB334_EXTENDED_M_CODE_UNIT_2_STA_0".M_code[113] OR "DB356_M_UNIT_2_STA_0".M_CODES_UNIT_2_STA_0.M113) AND NOT "DB356_M_UNIT_2_STA_0".M_CODES_UNIT_2_STA_0.Ack_M113 AND NOT "DB2120_MPP_ITC_IPC".RESET_FAULTS AND NOT "DB356_M_UNIT_2_STA_0".M_CODES_UNIT_2_STA_0.M_RESET_PULSE;
END_REGION

REGION Network 73: ACKNOWLEDGE M140- SWITCH ON ASPIRATION SYSTEM STATION 1 / ACKNOWLEDGE M85-LOAD-UNLOAD TRAP DOOR OPEN
   RUNG wire#powerrail
      Contact( "DB356_M_UNIT_2_STA_0".M_CODES_UNIT_2_STA_0.M140 )
      Contact( "DB1721_UNIT_02_STA_1_ASPIRATION_VALVE".SWITCH_ON )
      Coil( "DB356_M_UNIT_2_STA_0".M_CODES_UNIT_2_STA_0.Ack_M140 )
   END_RUNG
   // the same network as SCL:
   "DB356_M_UNIT_2_STA_0".M_CODES_UNIT_2_STA_0.Ack_M140 := "DB356_M_UNIT_2_STA_0".M_CODES_UNIT_2_STA_0.M140 AND "DB1721_UNIT_02_STA_1_ASPIRATION_VALVE".SWITCH_ON;
END_REGION

REGION Network 74: M140- SWITCH ON ASPIRATION SYSTEM STATION 1 / M85-LOAD-UNLOAD TRAP DOOR OPEN
   RUNG wire#powerrail
      Contact( "DB334_EXTENDED_M_CODE_UNIT_2_STA_0".M_code[140] )
      wire#w1
      I_Contact( "DB356_M_UNIT_2_STA_0".M_CODES_UNIT_2_STA_0.Ack_M140 )
      I_Contact( "DB2120_MPP_ITC_IPC".RESET_FAULTS )
      I_Contact( "DB356_M_UNIT_2_STA_0".M_CODES_UNIT_2_STA_0.M_RESET_PULSE )
      Coil( "DB356_M_UNIT_2_STA_0".M_CODES_UNIT_2_STA_0.M140 )
   END_RUNG
   RUNG wire#powerrail
      Contact( "DB356_M_UNIT_2_STA_0".M_CODES_UNIT_2_STA_0.M140 )
   END_RUNG wire#w1
   // the same network as SCL:
   "DB356_M_UNIT_2_STA_0".M_CODES_UNIT_2_STA_0.M140 := ("DB334_EXTENDED_M_CODE_UNIT_2_STA_0".M_code[140] OR "DB356_M_UNIT_2_STA_0".M_CODES_UNIT_2_STA_0.M140) AND NOT "DB356_M_UNIT_2_STA_0".M_CODES_UNIT_2_STA_0.Ack_M140 AND NOT "DB2120_MPP_ITC_IPC".RESET_FAULTS AND NOT "DB356_M_UNIT_2_STA_0".M_CODES_UNIT_2_STA_0.M_RESET_PULSE;
END_REGION

REGION Network 75: ACKNOWLEDGE M141- SWITCH OFF ASPIRATION SYSTEM STATION 1 / ACKNOWLEDGE M23-SWITCH ON SPINDLE FRAME BLOWING
   RUNG wire#powerrail
      Contact( "DB356_M_UNIT_2_STA_0".M_CODES_UNIT_2_STA_0.M141 )
      Contact( "DB1721_UNIT_02_STA_1_ASPIRATION_VALVE".SWITCH_OFF )
      Coil( "DB356_M_UNIT_2_STA_0".M_CODES_UNIT_2_STA_0.Ack_M141 )
   END_RUNG
   // the same network as SCL:
   "DB356_M_UNIT_2_STA_0".M_CODES_UNIT_2_STA_0.Ack_M141 := "DB356_M_UNIT_2_STA_0".M_CODES_UNIT_2_STA_0.M141 AND "DB1721_UNIT_02_STA_1_ASPIRATION_VALVE".SWITCH_OFF;
END_REGION

REGION Network 76: M141- SWITCH OFF ASPIRATION SYSTEM STATION 1 / M23-SWITCH ON SPINDLE FRAME BLOWING
   RUNG wire#powerrail
      Contact( "DB334_EXTENDED_M_CODE_UNIT_2_STA_0".M_code[141] )
      wire#w1
      I_Contact( "DB356_M_UNIT_2_STA_0".M_CODES_UNIT_2_STA_0.Ack_M141 )
      I_Contact( "DB2120_MPP_ITC_IPC".RESET_FAULTS )
      I_Contact( "DB356_M_UNIT_2_STA_0".M_CODES_UNIT_2_STA_0.M_RESET_PULSE )
      Coil( "DB356_M_UNIT_2_STA_0".M_CODES_UNIT_2_STA_0.M141 )
   END_RUNG
   RUNG wire#powerrail
      Contact( "DB356_M_UNIT_2_STA_0".M_CODES_UNIT_2_STA_0.M141 )
   END_RUNG wire#w1
   // the same network as SCL:
   "DB356_M_UNIT_2_STA_0".M_CODES_UNIT_2_STA_0.M141 := ("DB334_EXTENDED_M_CODE_UNIT_2_STA_0".M_code[141] OR "DB356_M_UNIT_2_STA_0".M_CODES_UNIT_2_STA_0.M141) AND NOT "DB356_M_UNIT_2_STA_0".M_CODES_UNIT_2_STA_0.Ack_M141 AND NOT "DB2120_MPP_ITC_IPC".RESET_FAULTS AND NOT "DB356_M_UNIT_2_STA_0".M_CODES_UNIT_2_STA_0.M_RESET_PULSE;
END_REGION

REGION Network 77: ACKNOWLEDGE M200-MAIN SAFETY DOOR, OPEN REQUEST (READ-IN DISABLE) / ACKNOWLEDGE M22-OPEN FRONT DOORS FOR TOOL CHANGE
   RUNG wire#powerrail
      Contact( "DB356_M_UNIT_2_STA_0".M_CODES_UNIT_2_STA_0.M200 )
      I_Contact( "DB7011_UNIT_2_MAIN_SAFETY_DOOR".SAFETY_DOOR.CLOSED_AND_LOCKED )
      Coil( "DB356_M_UNIT_2_STA_0".M_CODES_UNIT_2_STA_0.Ack_M200 )
   END_RUNG
   // the same network as SCL:
   "DB356_M_UNIT_2_STA_0".M_CODES_UNIT_2_STA_0.Ack_M200 := "DB356_M_UNIT_2_STA_0".M_CODES_UNIT_2_STA_0.M200 AND NOT "DB7011_UNIT_2_MAIN_SAFETY_DOOR".SAFETY_DOOR.CLOSED_AND_LOCKED;
END_REGION

REGION Network 78: M200-MAIN SAFETY DOOR, OPEN REQUEST (READ-IN DISABLE) / M22-OPEN FRONT DOORS FOR TOOL CHANGE
   RUNG wire#powerrail
      Contact( "DB334_EXTENDED_M_CODE_UNIT_2_STA_0".M_code[200] )
      wire#w1
      I_Contact( "DB356_M_UNIT_2_STA_0".M_CODES_UNIT_2_STA_0.Ack_M200 )
      I_Contact( "DB2120_MPP_ITC_IPC".RESET_FAULTS )
      wire#w2
      I_Contact( "DB356_M_UNIT_2_STA_0".M_CODES_UNIT_2_STA_0.M_RESET_PULSE )
      wire#w3
      Coil( "DB356_M_UNIT_2_STA_0".M_CODES_UNIT_2_STA_0.M200 )
   END_RUNG
   RUNG wire#powerrail
      Contact( "DB356_M_UNIT_2_STA_0".M_CODES_UNIT_2_STA_0.M200 )
   END_RUNG wire#w1
   RUNG wire#w2
      Contact( "DB7013_UNIT_2_STATION_4_SAFETY_DOOR".SAFETY_DOOR.CLOSED_AND_LOCKED )
   END_RUNG wire#w3
   // the same network as SCL:
   "DB356_M_UNIT_2_STA_0".M_CODES_UNIT_2_STA_0.M200 := ("DB334_EXTENDED_M_CODE_UNIT_2_STA_0".M_code[200] OR "DB356_M_UNIT_2_STA_0".M_CODES_UNIT_2_STA_0.M200) AND NOT "DB356_M_UNIT_2_STA_0".M_CODES_UNIT_2_STA_0.Ack_M200 AND NOT "DB2120_MPP_ITC_IPC".RESET_FAULTS AND (NOT "DB356_M_UNIT_2_STA_0".M_CODES_UNIT_2_STA_0.M_RESET_PULSE OR "DB7013_UNIT_2_STATION_4_SAFETY_DOOR".SAFETY_DOOR.CLOSED_AND_LOCKED);
END_REGION

REGION Network 79: ACKNOWLEDGE M201-SIDE R SAFETY DOOR, OPEN REQUEST (READ-IN DISABLE) / ACKNOWLEDGE M31-WAIT UPDATE TOOL
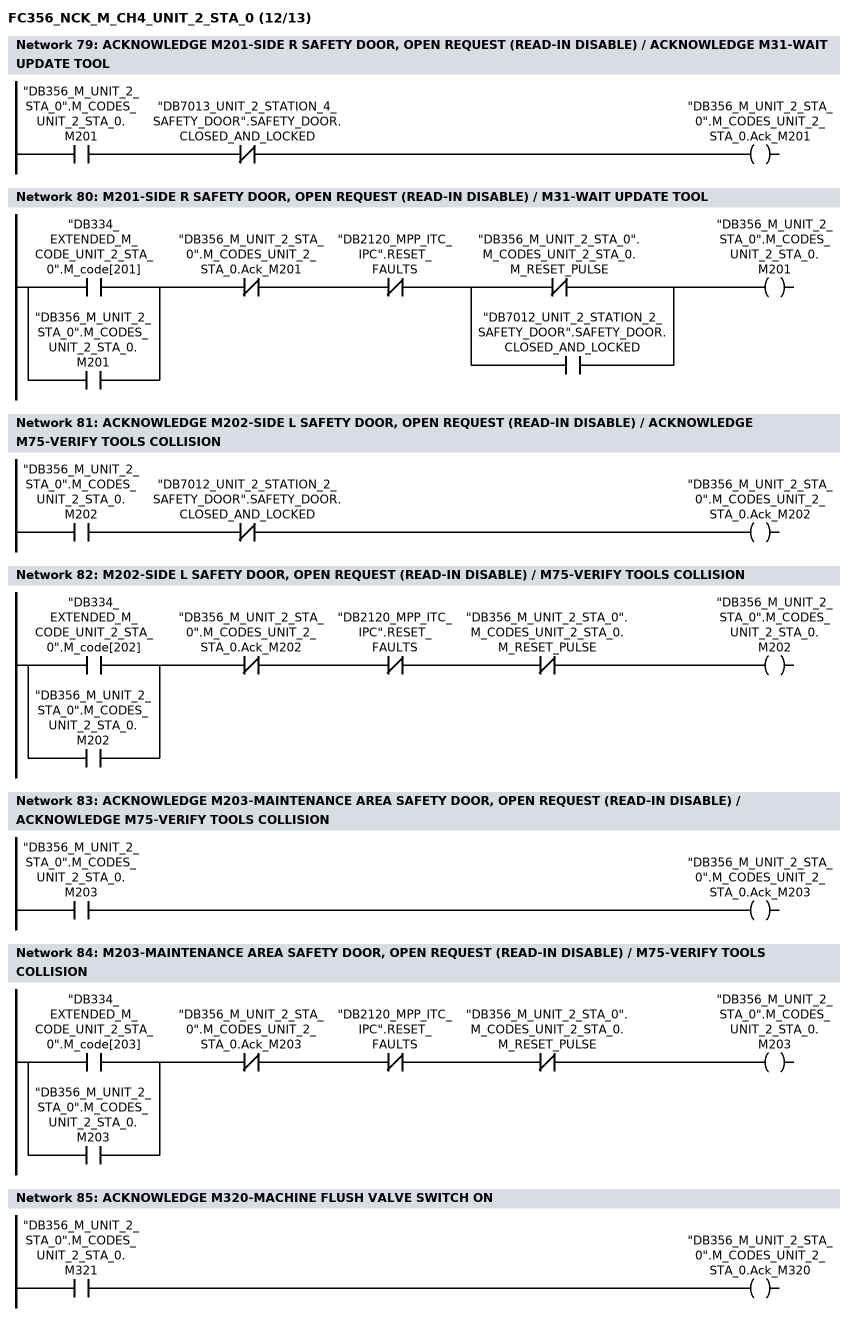
   RUNG wire#powerrail
      Contact( "DB356_M_UNIT_2_STA_0".M_CODES_UNIT_2_STA_0.M201 )
      I_Contact( "DB7013_UNIT_2_STATION_4_SAFETY_DOOR".SAFETY_DOOR.CLOSED_AND_LOCKED )
      Coil( "DB356_M_UNIT_2_STA_0".M_CODES_UNIT_2_STA_0.Ack_M201 )
   END_RUNG
   // the same network as SCL:
   "DB356_M_UNIT_2_STA_0".M_CODES_UNIT_2_STA_0.Ack_M201 := "DB356_M_UNIT_2_STA_0".M_CODES_UNIT_2_STA_0.M201 AND NOT "DB7013_UNIT_2_STATION_4_SAFETY_DOOR".SAFETY_DOOR.CLOSED_AND_LOCKED;
END_REGION

REGION Network 80: M201-SIDE R SAFETY DOOR, OPEN REQUEST (READ-IN DISABLE) / M31-WAIT UPDATE TOOL
   RUNG wire#powerrail
      Contact( "DB334_EXTENDED_M_CODE_UNIT_2_STA_0".M_code[201] )
      wire#w1
      I_Contact( "DB356_M_UNIT_2_STA_0".M_CODES_UNIT_2_STA_0.Ack_M201 )
      I_Contact( "DB2120_MPP_ITC_IPC".RESET_FAULTS )
      wire#w2
      I_Contact( "DB356_M_UNIT_2_STA_0".M_CODES_UNIT_2_STA_0.M_RESET_PULSE )
      wire#w3
      Coil( "DB356_M_UNIT_2_STA_0".M_CODES_UNIT_2_STA_0.M201 )
   END_RUNG
   RUNG wire#powerrail
      Contact( "DB356_M_UNIT_2_STA_0".M_CODES_UNIT_2_STA_0.M201 )
   END_RUNG wire#w1
   RUNG wire#w2
      Contact( "DB7012_UNIT_2_STATION_2_SAFETY_DOOR".SAFETY_DOOR.CLOSED_AND_LOCKED )
   END_RUNG wire#w3
   // the same network as SCL:
   "DB356_M_UNIT_2_STA_0".M_CODES_UNIT_2_STA_0.M201 := ("DB334_EXTENDED_M_CODE_UNIT_2_STA_0".M_code[201] OR "DB356_M_UNIT_2_STA_0".M_CODES_UNIT_2_STA_0.M201) AND NOT "DB356_M_UNIT_2_STA_0".M_CODES_UNIT_2_STA_0.Ack_M201 AND NOT "DB2120_MPP_ITC_IPC".RESET_FAULTS AND (NOT "DB356_M_UNIT_2_STA_0".M_CODES_UNIT_2_STA_0.M_RESET_PULSE OR "DB7012_UNIT_2_STATION_2_SAFETY_DOOR".SAFETY_DOOR.CLOSED_AND_LOCKED);
END_REGION

REGION Network 81: ACKNOWLEDGE M202-SIDE L SAFETY DOOR, OPEN REQUEST (READ-IN DISABLE) / ACKNOWLEDGE M75-VERIFY TOOLS COLLISION
   RUNG wire#powerrail
      Contact( "DB356_M_UNIT_2_STA_0".M_CODES_UNIT_2_STA_0.M202 )
      I_Contact( "DB7012_UNIT_2_STATION_2_SAFETY_DOOR".SAFETY_DOOR.CLOSED_AND_LOCKED )
      Coil( "DB356_M_UNIT_2_STA_0".M_CODES_UNIT_2_STA_0.Ack_M202 )
   END_RUNG
   // the same network as SCL:
   "DB356_M_UNIT_2_STA_0".M_CODES_UNIT_2_STA_0.Ack_M202 := "DB356_M_UNIT_2_STA_0".M_CODES_UNIT_2_STA_0.M202 AND NOT "DB7012_UNIT_2_STATION_2_SAFETY_DOOR".SAFETY_DOOR.CLOSED_AND_LOCKED;
END_REGION

REGION Network 82: M202-SIDE L SAFETY DOOR, OPEN REQUEST (READ-IN DISABLE) / M75-VERIFY TOOLS COLLISION
   RUNG wire#powerrail
      Contact( "DB334_EXTENDED_M_CODE_UNIT_2_STA_0".M_code[202] )
      wire#w1
      I_Contact( "DB356_M_UNIT_2_STA_0".M_CODES_UNIT_2_STA_0.Ack_M202 )
      I_Contact( "DB2120_MPP_ITC_IPC".RESET_FAULTS )
      I_Contact( "DB356_M_UNIT_2_STA_0".M_CODES_UNIT_2_STA_0.M_RESET_PULSE )
      Coil( "DB356_M_UNIT_2_STA_0".M_CODES_UNIT_2_STA_0.M202 )
   END_RUNG
   RUNG wire#powerrail
      Contact( "DB356_M_UNIT_2_STA_0".M_CODES_UNIT_2_STA_0.M202 )
   END_RUNG wire#w1
   // the same network as SCL:
   "DB356_M_UNIT_2_STA_0".M_CODES_UNIT_2_STA_0.M202 := ("DB334_EXTENDED_M_CODE_UNIT_2_STA_0".M_code[202] OR "DB356_M_UNIT_2_STA_0".M_CODES_UNIT_2_STA_0.M202) AND NOT "DB356_M_UNIT_2_STA_0".M_CODES_UNIT_2_STA_0.Ack_M202 AND NOT "DB2120_MPP_ITC_IPC".RESET_FAULTS AND NOT "DB356_M_UNIT_2_STA_0".M_CODES_UNIT_2_STA_0.M_RESET_PULSE;
END_REGION

REGION Network 83: ACKNOWLEDGE M203-MAINTENANCE AREA SAFETY DOOR, OPEN REQUEST (READ-IN DISABLE) / ACKNOWLEDGE M75-VERIFY TOOLS COLLISION
   RUNG wire#powerrail
      Contact( "DB356_M_UNIT_2_STA_0".M_CODES_UNIT_2_STA_0.M203 )
      Coil( "DB356_M_UNIT_2_STA_0".M_CODES_UNIT_2_STA_0.Ack_M203 )
   END_RUNG
   // the same network as SCL:
   "DB356_M_UNIT_2_STA_0".M_CODES_UNIT_2_STA_0.Ack_M203 := "DB356_M_UNIT_2_STA_0".M_CODES_UNIT_2_STA_0.M203;
END_REGION

REGION Network 84: M203-MAINTENANCE AREA SAFETY DOOR, OPEN REQUEST (READ-IN DISABLE) / M75-VERIFY TOOLS COLLISION
   RUNG wire#powerrail
      Contact( "DB334_EXTENDED_M_CODE_UNIT_2_STA_0".M_code[203] )
      wire#w1
      I_Contact( "DB356_M_UNIT_2_STA_0".M_CODES_UNIT_2_STA_0.Ack_M203 )
      I_Contact( "DB2120_MPP_ITC_IPC".RESET_FAULTS )
      I_Contact( "DB356_M_UNIT_2_STA_0".M_CODES_UNIT_2_STA_0.M_RESET_PULSE )
      Coil( "DB356_M_UNIT_2_STA_0".M_CODES_UNIT_2_STA_0.M203 )
   END_RUNG
   RUNG wire#powerrail
      Contact( "DB356_M_UNIT_2_STA_0".M_CODES_UNIT_2_STA_0.M203 )
   END_RUNG wire#w1
   // the same network as SCL:
   "DB356_M_UNIT_2_STA_0".M_CODES_UNIT_2_STA_0.M203 := ("DB334_EXTENDED_M_CODE_UNIT_2_STA_0".M_code[203] OR "DB356_M_UNIT_2_STA_0".M_CODES_UNIT_2_STA_0.M203) AND NOT "DB356_M_UNIT_2_STA_0".M_CODES_UNIT_2_STA_0.Ack_M203 AND NOT "DB2120_MPP_ITC_IPC".RESET_FAULTS AND NOT "DB356_M_UNIT_2_STA_0".M_CODES_UNIT_2_STA_0.M_RESET_PULSE;
END_REGION

REGION Network 85: ACKNOWLEDGE M320-MACHINE FLUSH VALVE SWITCH ON
   RUNG wire#powerrail
      Contact( "DB356_M_UNIT_2_STA_0".M_CODES_UNIT_2_STA_0.M321 )
      Coil( "DB356_M_UNIT_2_STA_0".M_CODES_UNIT_2_STA_0.Ack_M320 )
   END_RUNG
   // the same network as SCL:
   "DB356_M_UNIT_2_STA_0".M_CODES_UNIT_2_STA_0.Ack_M320 := "DB356_M_UNIT_2_STA_0".M_CODES_UNIT_2_STA_0.M321;
END_REGION

REGION Network 86: READ-IN DISABLE / Read-in disable
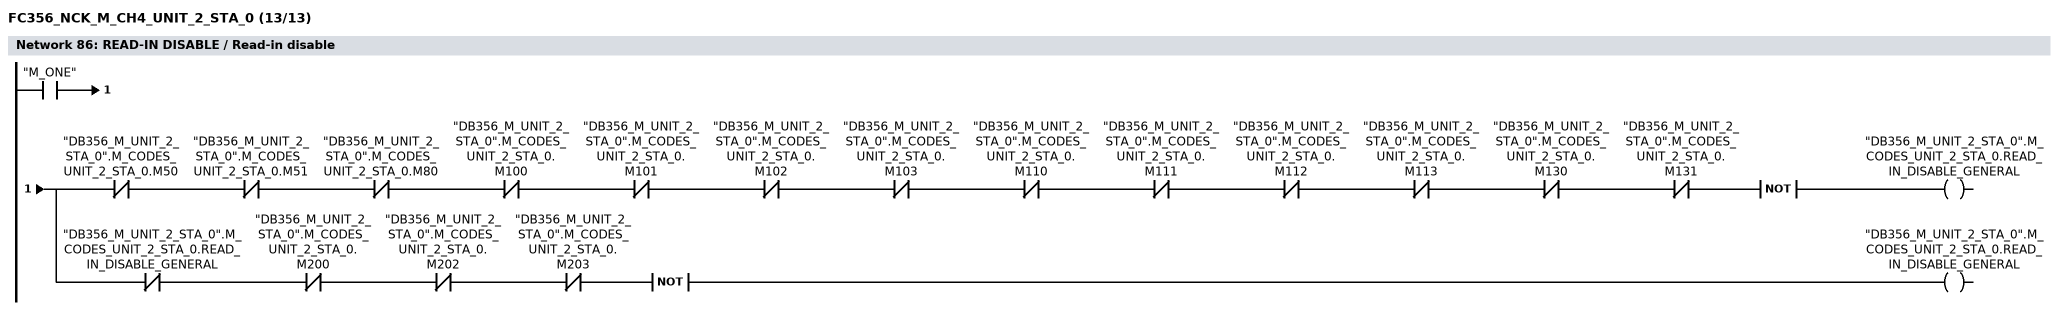
   RUNG wire#powerrail
      Contact( "M_ONE" )
      wire#w1
      I_Contact( "DB356_M_UNIT_2_STA_0".M_CODES_UNIT_2_STA_0.M50 )
      I_Contact( "DB356_M_UNIT_2_STA_0".M_CODES_UNIT_2_STA_0.M51 )
      I_Contact( "DB356_M_UNIT_2_STA_0".M_CODES_UNIT_2_STA_0.M80 )
      I_Contact( "DB356_M_UNIT_2_STA_0".M_CODES_UNIT_2_STA_0.M100 )
      I_Contact( "DB356_M_UNIT_2_STA_0".M_CODES_UNIT_2_STA_0.M101 )
      I_Contact( "DB356_M_UNIT_2_STA_0".M_CODES_UNIT_2_STA_0.M102 )
      I_Contact( "DB356_M_UNIT_2_STA_0".M_CODES_UNIT_2_STA_0.M103 )
      I_Contact( "DB356_M_UNIT_2_STA_0".M_CODES_UNIT_2_STA_0.M110 )
      I_Contact( "DB356_M_UNIT_2_STA_0".M_CODES_UNIT_2_STA_0.M111 )
      I_Contact( "DB356_M_UNIT_2_STA_0".M_CODES_UNIT_2_STA_0.M112 )
      I_Contact( "DB356_M_UNIT_2_STA_0".M_CODES_UNIT_2_STA_0.M113 )
      I_Contact( "DB356_M_UNIT_2_STA_0".M_CODES_UNIT_2_STA_0.M130 )
      I_Contact( "DB356_M_UNIT_2_STA_0".M_CODES_UNIT_2_STA_0.M131 )
      Not()
      Coil( "DB356_M_UNIT_2_STA_0".M_CODES_UNIT_2_STA_0.READ_IN_DISABLE_GENERAL )
   END_RUNG
   RUNG wire#w1
      I_Contact( "DB356_M_UNIT_2_STA_0".M_CODES_UNIT_2_STA_0.READ_IN_DISABLE_GENERAL )
      I_Contact( "DB356_M_UNIT_2_STA_0".M_CODES_UNIT_2_STA_0.M200 )
      I_Contact( "DB356_M_UNIT_2_STA_0".M_CODES_UNIT_2_STA_0.M202 )
      I_Contact( "DB356_M_UNIT_2_STA_0".M_CODES_UNIT_2_STA_0.M203 )
      Not()
      Coil( "DB356_M_UNIT_2_STA_0".M_CODES_UNIT_2_STA_0.READ_IN_DISABLE_GENERAL )
   END_RUNG
   // the same network as SCL:
   "DB356_M_UNIT_2_STA_0".M_CODES_UNIT_2_STA_0.READ_IN_DISABLE_GENERAL := NOT ("M_ONE" AND NOT "DB356_M_UNIT_2_STA_0".M_CODES_UNIT_2_STA_0.M50 AND NOT "DB356_M_UNIT_2_STA_0".M_CODES_UNIT_2_STA_0.M51 AND NOT "DB356_M_UNIT_2_STA_0".M_CODES_UNIT_2_STA_0.M80 AND NOT "DB356_M_UNIT_2_STA_0".M_CODES_UNIT_2_STA_0.M100 AND NOT "DB356_M_UNIT_2_STA_0".M_CODES_UNIT_2_STA_0.M101 AND NOT "DB356_M_UNIT_2_STA_0".M_CODES_UNIT_2_STA_0.M102 AND NOT "DB356_M_UNIT_2_STA_0".M_CODES_UNIT_2_STA_0.M103 AND NOT "DB356_M_UNIT_2_STA_0".M_CODES_UNIT_2_STA_0.M110 AND NOT "DB356_M_UNIT_2_STA_0".M_CODES_UNIT_2_STA_0.M111 AND NOT "DB356_M_UNIT_2_STA_0".M_CODES_UNIT_2_STA_0.M112 AND NOT "DB356_M_UNIT_2_STA_0".M_CODES_UNIT_2_STA_0.M113 AND NOT "DB356_M_UNIT_2_STA_0".M_CODES_UNIT_2_STA_0.M130 AND NOT "DB356_M_UNIT_2_STA_0".M_CODES_UNIT_2_STA_0.M131);
   "DB356_M_UNIT_2_STA_0".M_CODES_UNIT_2_STA_0.READ_IN_DISABLE_GENERAL := NOT ("M_ONE" AND NOT "DB356_M_UNIT_2_STA_0".M_CODES_UNIT_2_STA_0.READ_IN_DISABLE_GENERAL AND NOT "DB356_M_UNIT_2_STA_0".M_CODES_UNIT_2_STA_0.M200 AND NOT "DB356_M_UNIT_2_STA_0".M_CODES_UNIT_2_STA_0.M202 AND NOT "DB356_M_UNIT_2_STA_0".M_CODES_UNIT_2_STA_0.M203);
END_REGION
END_FUNCTION
